REGION Network 38: ABFV 207 OPEN FB
   RUNG wire#powerrail
      { S7_Templates := "SrcType := Int" } EQ_Contact(in1 := "MODE SELECTION DB"."UF PLC_1 MODE BUFF", in2 := 1)
      { S7_Templates := "SrcType := Int" } EQ_Contact(in1 := "MODE SELECTION DB"."UF PLC_1 PROCESS BUFF", in2 := 870)
      Contact( "INPUT MAPPING DB"."ABFV-207 FEED BACK OPEN" )
      Move(in := 875, out1 => "MODE SELECTION DB"."UF PLC_1 PROCESS BUFF")
   END_RUNG
   // the same network as SCL:
   IF ("MODE SELECTION DB"."UF PLC_1 MODE BUFF" = 1) AND ("MODE SELECTION DB"."UF PLC_1 PROCESS BUFF" = 870) AND "INPUT MAPPING DB"."ABFV-207 FEED BACK OPEN" THEN
       "MODE SELECTION DB"."UF PLC_1 PROCESS BUFF" := 875;
   END_IF;
END_REGION

REGION Network 39: ABFV 208 OPEN FB
   RUNG wire#powerrail
      { S7_Templates := "SrcType := Int" } EQ_Contact(in1 := "MODE SELECTION DB"."UF PLC_1 MODE BUFF", in2 := 1)
      { S7_Templates := "SrcType := Int" } EQ_Contact(in1 := "MODE SELECTION DB"."UF PLC_1 PROCESS BUFF", in2 := 875)
      Contact( "INPUT MAPPING DB"."ABFV-208 FEED BACK OPEN" )
      { S7_Templates := "time_type := Time" } "IEC_Timer_0_DB_85".TON(pt := T#5s, et =>)
      Move(in := 880, out1 => "MODE SELECTION DB"."UF PLC_1 PROCESS BUFF")
   END_RUNG
   // the same network as SCL:
   "IEC_Timer_0_DB_85".TON(IN := ("MODE SELECTION DB"."UF PLC_1 MODE BUFF" = 1) AND ("MODE SELECTION DB"."UF PLC_1 PROCESS BUFF" = 875) AND "INPUT MAPPING DB"."ABFV-208 FEED BACK OPEN",
                           PT := T#5s);
   IF "IEC_Timer_0_DB_85".Q THEN "MODE SELECTION DB"."UF PLC_1 PROCESS BUFF" := 880; END_IF;
END_REGION

REGION Network 40: BACKWASH_1
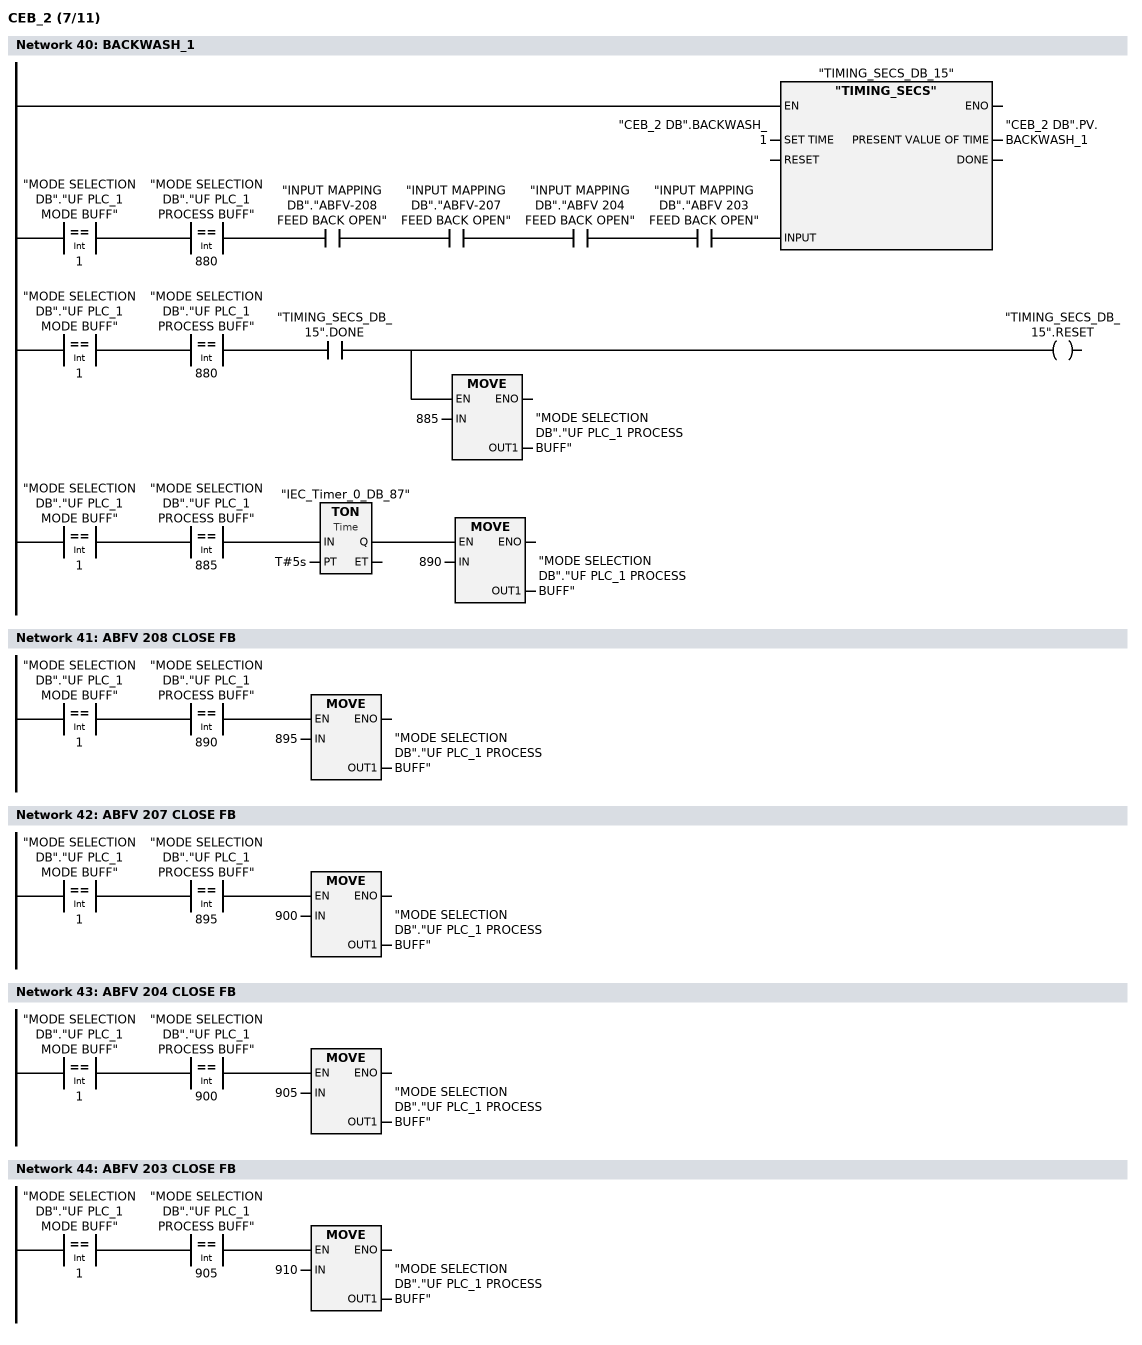
   RUNG wire#powerrail
      "TIMING_SECS_DB_15"(INPUT := wire#w1, "SET TIME" := "CEB_2 DB".BACKWASH_1, RESET :=, "PRESENT VALUE OF TIME" => "CEB_2 DB".PV.BACKWASH_1, DONE =>)
   END_RUNG
   RUNG wire#powerrail
      { S7_Templates := "SrcType := Int" } EQ_Contact(in1 := "MODE SELECTION DB"."UF PLC_1 MODE BUFF", in2 := 1)
      { S7_Templates := "SrcType := Int" } EQ_Contact(in1 := "MODE SELECTION DB"."UF PLC_1 PROCESS BUFF", in2 := 880)
      Contact( "INPUT MAPPING DB"."ABFV-208 FEED BACK OPEN" )
      Contact( "INPUT MAPPING DB"."ABFV-207 FEED BACK OPEN" )
      Contact( "INPUT MAPPING DB"."ABFV 204 FEED BACK OPEN" )
      Contact( "INPUT MAPPING DB"."ABFV 203 FEED BACK OPEN" )
   END_RUNG wire#w1
   RUNG wire#powerrail
      { S7_Templates := "SrcType := Int" } EQ_Contact(in1 := "MODE SELECTION DB"."UF PLC_1 MODE BUFF", in2 := 1)
      { S7_Templates := "SrcType := Int" } EQ_Contact(in1 := "MODE SELECTION DB"."UF PLC_1 PROCESS BUFF", in2 := 880)
      Contact( "TIMING_SECS_DB_15".DONE )
      wire#w2
      Coil( "TIMING_SECS_DB_15".RESET )
   END_RUNG
   RUNG wire#w2
      Move(in := 885, out1 => "MODE SELECTION DB"."UF PLC_1 PROCESS BUFF")
   END_RUNG
   RUNG wire#powerrail
      { S7_Templates := "SrcType := Int" } EQ_Contact(in1 := "MODE SELECTION DB"."UF PLC_1 MODE BUFF", in2 := 1)
      { S7_Templates := "SrcType := Int" } EQ_Contact(in1 := "MODE SELECTION DB"."UF PLC_1 PROCESS BUFF", in2 := 885)
      { S7_Templates := "time_type := Time" } "IEC_Timer_0_DB_87".TON(pt := T#5s, et =>)
      Move(in := 890, out1 => "MODE SELECTION DB"."UF PLC_1 PROCESS BUFF")
   END_RUNG
   // the same network as SCL:
   "TIMING_SECS_DB_15"("SET TIME" := "CEB_2 DB".BACKWASH_1,   // "TIMING_SECS"
                       INPUT := ("MODE SELECTION DB"."UF PLC_1 MODE BUFF" = 1) AND ("MODE SELECTION DB"."UF PLC_1 PROCESS BUFF" = 880) AND "INPUT MAPPING DB"."ABFV-208 FEED BACK OPEN" AND "INPUT MAPPING DB"."ABFV-207 FEED BACK OPEN" AND "INPUT MAPPING DB"."ABFV 204 FEED BACK OPEN" AND "INPUT MAPPING DB"."ABFV 203 FEED BACK OPEN",
                       "PRESENT VALUE OF TIME" => "CEB_2 DB".PV.BACKWASH_1);
   "TIMING_SECS_DB_15".RESET := ("MODE SELECTION DB"."UF PLC_1 MODE BUFF" = 1) AND ("MODE SELECTION DB"."UF PLC_1 PROCESS BUFF" = 880) AND "TIMING_SECS_DB_15".DONE;
   IF "TIMING_SECS_DB_15".RESET THEN "MODE SELECTION DB"."UF PLC_1 PROCESS BUFF" := 885; END_IF;
   "IEC_Timer_0_DB_87".TON(IN := ("MODE SELECTION DB"."UF PLC_1 MODE BUFF" = 1) AND ("MODE SELECTION DB"."UF PLC_1 PROCESS BUFF" = 885),
                           PT := T#5s);
   IF "IEC_Timer_0_DB_87".Q THEN "MODE SELECTION DB"."UF PLC_1 PROCESS BUFF" := 890; END_IF;
END_REGION

REGION Network 41: ABFV 208 CLOSE FB
   RUNG wire#powerrail
      { S7_Templates := "SrcType := Int" } EQ_Contact(in1 := "MODE SELECTION DB"."UF PLC_1 MODE BUFF", in2 := 1)
      { S7_Templates := "SrcType := Int" } EQ_Contact(in1 := "MODE SELECTION DB"."UF PLC_1 PROCESS BUFF", in2 := 890)
      Move(in := 895, out1 => "MODE SELECTION DB"."UF PLC_1 PROCESS BUFF")
   END_RUNG
   // the same network as SCL:
   IF ("MODE SELECTION DB"."UF PLC_1 MODE BUFF" = 1) AND ("MODE SELECTION DB"."UF PLC_1 PROCESS BUFF" = 890) THEN
       "MODE SELECTION DB"."UF PLC_1 PROCESS BUFF" := 895;
   END_IF;
END_REGION

REGION Network 42: ABFV 207 CLOSE FB
   RUNG wire#powerrail
      { S7_Templates := "SrcType := Int" } EQ_Contact(in1 := "MODE SELECTION DB"."UF PLC_1 MODE BUFF", in2 := 1)
      { S7_Templates := "SrcType := Int" } EQ_Contact(in1 := "MODE SELECTION DB"."UF PLC_1 PROCESS BUFF", in2 := 895)
      Move(in := 900, out1 => "MODE SELECTION DB"."UF PLC_1 PROCESS BUFF")
   END_RUNG
   // the same network as SCL:
   IF ("MODE SELECTION DB"."UF PLC_1 MODE BUFF" = 1) AND ("MODE SELECTION DB"."UF PLC_1 PROCESS BUFF" = 895) THEN
       "MODE SELECTION DB"."UF PLC_1 PROCESS BUFF" := 900;
   END_IF;
END_REGION

REGION Network 43: ABFV 204 CLOSE FB
   RUNG wire#powerrail
      { S7_Templates := "SrcType := Int" } EQ_Contact(in1 := "MODE SELECTION DB"."UF PLC_1 MODE BUFF", in2 := 1)
      { S7_Templates := "SrcType := Int" } EQ_Contact(in1 := "MODE SELECTION DB"."UF PLC_1 PROCESS BUFF", in2 := 900)
      Move(in := 905, out1 => "MODE SELECTION DB"."UF PLC_1 PROCESS BUFF")
   END_RUNG
   // the same network as SCL:
   IF ("MODE SELECTION DB"."UF PLC_1 MODE BUFF" = 1) AND ("MODE SELECTION DB"."UF PLC_1 PROCESS BUFF" = 900) THEN
       "MODE SELECTION DB"."UF PLC_1 PROCESS BUFF" := 905;
   END_IF;
END_REGION

REGION Network 44: ABFV 203 CLOSE FB
   RUNG wire#powerrail
      { S7_Templates := "SrcType := Int" } EQ_Contact(in1 := "MODE SELECTION DB"."UF PLC_1 MODE BUFF", in2 := 1)
      { S7_Templates := "SrcType := Int" } EQ_Contact(in1 := "MODE SELECTION DB"."UF PLC_1 PROCESS BUFF", in2 := 905)
      Move(in := 910, out1 => "MODE SELECTION DB"."UF PLC_1 PROCESS BUFF")
   END_RUNG
   // the same network as SCL:
   IF ("MODE SELECTION DB"."UF PLC_1 MODE BUFF" = 1) AND ("MODE SELECTION DB"."UF PLC_1 PROCESS BUFF" = 905) THEN
       "MODE SELECTION DB"."UF PLC_1 PROCESS BUFF" := 910;
   END_IF;
END_REGION

REGION Network 45: 915
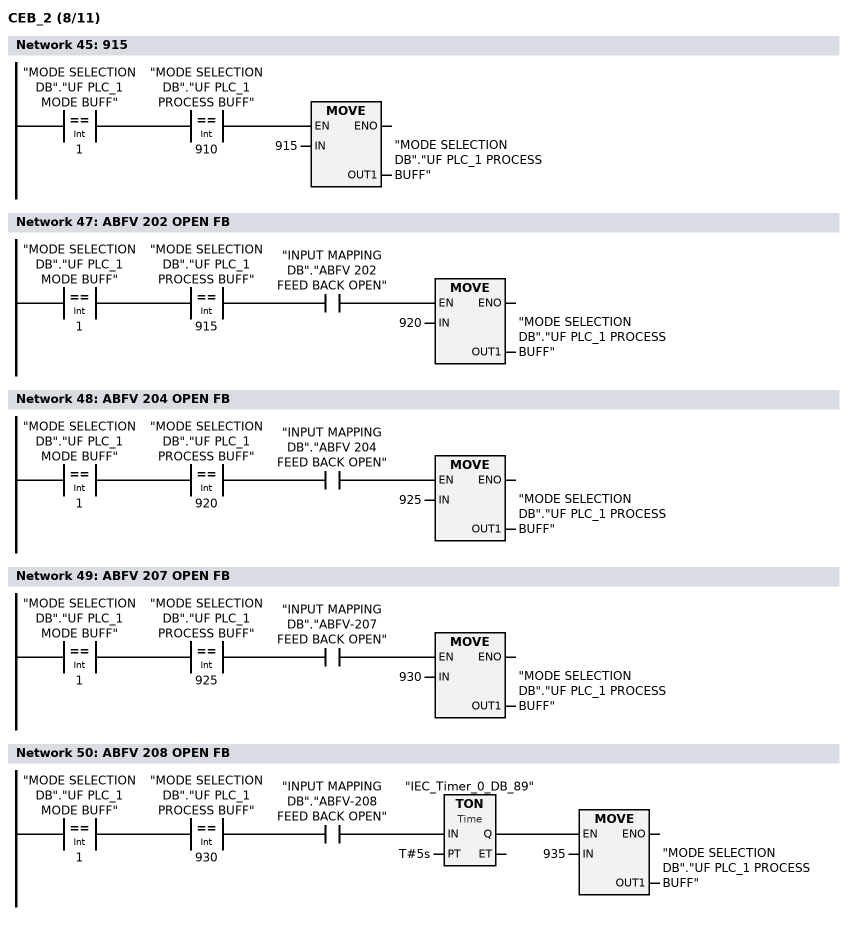
   RUNG wire#powerrail
      { S7_Templates := "SrcType := Int" } EQ_Contact(in1 := "MODE SELECTION DB"."UF PLC_1 MODE BUFF", in2 := 1)
      { S7_Templates := "SrcType := Int" } EQ_Contact(in1 := "MODE SELECTION DB"."UF PLC_1 PROCESS BUFF", in2 := 910)
      Move(in := 915, out1 => "MODE SELECTION DB"."UF PLC_1 PROCESS BUFF")
   END_RUNG
   // the same network as SCL:
   IF ("MODE SELECTION DB"."UF PLC_1 MODE BUFF" = 1) AND ("MODE SELECTION DB"."UF PLC_1 PROCESS BUFF" = 910) THEN
       "MODE SELECTION DB"."UF PLC_1 PROCESS BUFF" := 915;
   END_IF;
END_REGION

REGION Network 47: ABFV 202 OPEN FB
   RUNG wire#powerrail
      { S7_Templates := "SrcType := Int" } EQ_Contact(in1 := "MODE SELECTION DB"."UF PLC_1 MODE BUFF", in2 := 1)
      { S7_Templates := "SrcType := Int" } EQ_Contact(in1 := "MODE SELECTION DB"."UF PLC_1 PROCESS BUFF", in2 := 915)
      Contact( "INPUT MAPPING DB"."ABFV 202 FEED BACK OPEN" )
      Move(in := 920, out1 => "MODE SELECTION DB"."UF PLC_1 PROCESS BUFF")
   END_RUNG
   // the same network as SCL:
   IF ("MODE SELECTION DB"."UF PLC_1 MODE BUFF" = 1) AND ("MODE SELECTION DB"."UF PLC_1 PROCESS BUFF" = 915) AND "INPUT MAPPING DB"."ABFV 202 FEED BACK OPEN" THEN
       "MODE SELECTION DB"."UF PLC_1 PROCESS BUFF" := 920;
   END_IF;
END_REGION

REGION Network 48: ABFV 204 OPEN FB
   RUNG wire#powerrail
      { S7_Templates := "SrcType := Int" } EQ_Contact(in1 := "MODE SELECTION DB"."UF PLC_1 MODE BUFF", in2 := 1)
      { S7_Templates := "SrcType := Int" } EQ_Contact(in1 := "MODE SELECTION DB"."UF PLC_1 PROCESS BUFF", in2 := 920)
      Contact( "INPUT MAPPING DB"."ABFV 204 FEED BACK OPEN" )
      Move(in := 925, out1 => "MODE SELECTION DB"."UF PLC_1 PROCESS BUFF")
   END_RUNG
   // the same network as SCL:
   IF ("MODE SELECTION DB"."UF PLC_1 MODE BUFF" = 1) AND ("MODE SELECTION DB"."UF PLC_1 PROCESS BUFF" = 920) AND "INPUT MAPPING DB"."ABFV 204 FEED BACK OPEN" THEN
       "MODE SELECTION DB"."UF PLC_1 PROCESS BUFF" := 925;
   END_IF;
END_REGION

REGION Network 49: ABFV 207 OPEN FB
   RUNG wire#powerrail
      { S7_Templates := "SrcType := Int" } EQ_Contact(in1 := "MODE SELECTION DB"."UF PLC_1 MODE BUFF", in2 := 1)
      { S7_Templates := "SrcType := Int" } EQ_Contact(in1 := "MODE SELECTION DB"."UF PLC_1 PROCESS BUFF", in2 := 925)
      Contact( "INPUT MAPPING DB"."ABFV-207 FEED BACK OPEN" )
      Move(in := 930, out1 => "MODE SELECTION DB"."UF PLC_1 PROCESS BUFF")
   END_RUNG
   // the same network as SCL:
   IF ("MODE SELECTION DB"."UF PLC_1 MODE BUFF" = 1) AND ("MODE SELECTION DB"."UF PLC_1 PROCESS BUFF" = 925) AND "INPUT MAPPING DB"."ABFV-207 FEED BACK OPEN" THEN
       "MODE SELECTION DB"."UF PLC_1 PROCESS BUFF" := 930;
   END_IF;
END_REGION

REGION Network 50: ABFV 208 OPEN FB
   RUNG wire#powerrail
      { S7_Templates := "SrcType := Int" } EQ_Contact(in1 := "MODE SELECTION DB"."UF PLC_1 MODE BUFF", in2 := 1)
      { S7_Templates := "SrcType := Int" } EQ_Contact(in1 := "MODE SELECTION DB"."UF PLC_1 PROCESS BUFF", in2 := 930)
      Contact( "INPUT MAPPING DB"."ABFV-208 FEED BACK OPEN" )
      { S7_Templates := "time_type := Time" } "IEC_Timer_0_DB_89".TON(pt := T#5s, et =>)
      Move(in := 935, out1 => "MODE SELECTION DB"."UF PLC_1 PROCESS BUFF")
   END_RUNG
   // the same network as SCL:
   "IEC_Timer_0_DB_89".TON(IN := ("MODE SELECTION DB"."UF PLC_1 MODE BUFF" = 1) AND ("MODE SELECTION DB"."UF PLC_1 PROCESS BUFF" = 930) AND "INPUT MAPPING DB"."ABFV-208 FEED BACK OPEN",
                           PT := T#5s);
   IF "IEC_Timer_0_DB_89".Q THEN "MODE SELECTION DB"."UF PLC_1 PROCESS BUFF" := 935; END_IF;
END_REGION

REGION Network 51: BACKWASH_2
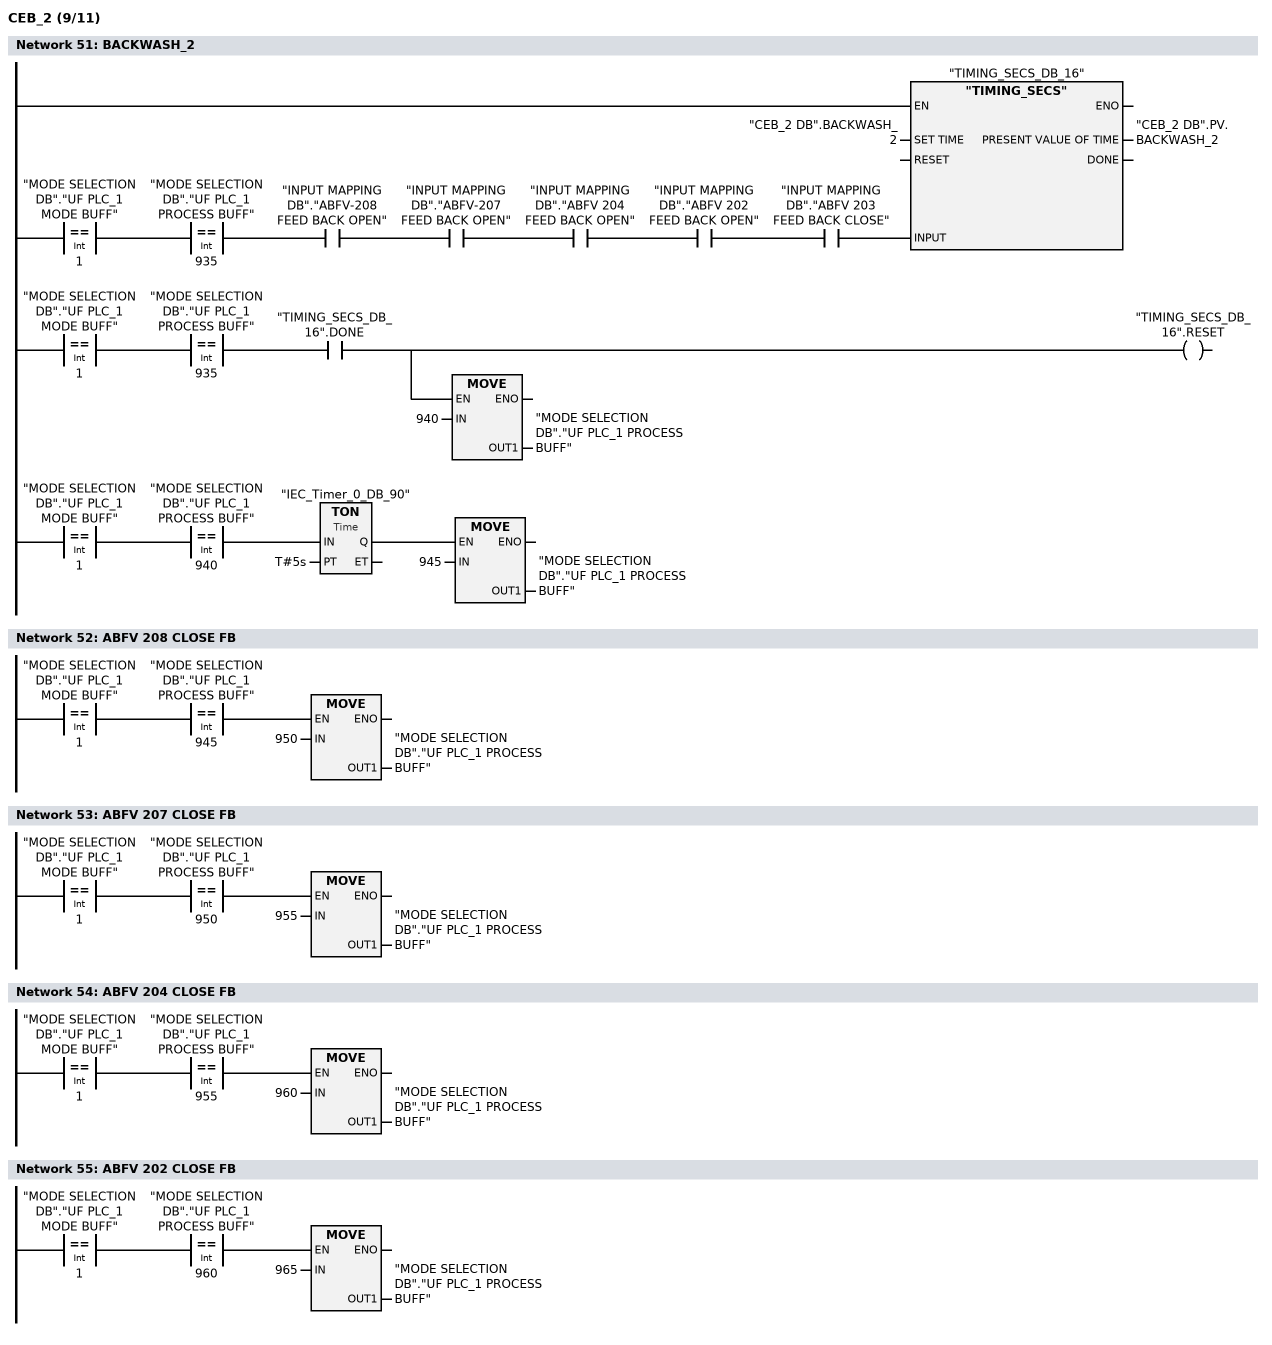
   RUNG wire#powerrail
      "TIMING_SECS_DB_16"(INPUT := wire#w1, "SET TIME" := "CEB_2 DB".BACKWASH_2, RESET :=, "PRESENT VALUE OF TIME" => "CEB_2 DB".PV.BACKWASH_2, DONE =>)
   END_RUNG
   RUNG wire#powerrail
      { S7_Templates := "SrcType := Int" } EQ_Contact(in1 := "MODE SELECTION DB"."UF PLC_1 MODE BUFF", in2 := 1)
      { S7_Templates := "SrcType := Int" } EQ_Contact(in1 := "MODE SELECTION DB"."UF PLC_1 PROCESS BUFF", in2 := 935)
      Contact( "INPUT MAPPING DB"."ABFV-208 FEED BACK OPEN" )
      Contact( "INPUT MAPPING DB"."ABFV-207 FEED BACK OPEN" )
      Contact( "INPUT MAPPING DB"."ABFV 204 FEED BACK OPEN" )
      Contact( "INPUT MAPPING DB"."ABFV 202 FEED BACK OPEN" )
      Contact( "INPUT MAPPING DB"."ABFV 203 FEED BACK CLOSE" )
   END_RUNG wire#w1
   RUNG wire#powerrail
      { S7_Templates := "SrcType := Int" } EQ_Contact(in1 := "MODE SELECTION DB"."UF PLC_1 MODE BUFF", in2 := 1)
      { S7_Templates := "SrcType := Int" } EQ_Contact(in1 := "MODE SELECTION DB"."UF PLC_1 PROCESS BUFF", in2 := 935)
      Contact( "TIMING_SECS_DB_16".DONE )
      wire#w2
      Coil( "TIMING_SECS_DB_16".RESET )
   END_RUNG
   RUNG wire#w2
      Move(in := 940, out1 => "MODE SELECTION DB"."UF PLC_1 PROCESS BUFF")
   END_RUNG
   RUNG wire#powerrail
      { S7_Templates := "SrcType := Int" } EQ_Contact(in1 := "MODE SELECTION DB"."UF PLC_1 MODE BUFF", in2 := 1)
      { S7_Templates := "SrcType := Int" } EQ_Contact(in1 := "MODE SELECTION DB"."UF PLC_1 PROCESS BUFF", in2 := 940)
      { S7_Templates := "time_type := Time" } "IEC_Timer_0_DB_90".TON(pt := T#5s, et =>)
      Move(in := 945, out1 => "MODE SELECTION DB"."UF PLC_1 PROCESS BUFF")
   END_RUNG
   // the same network as SCL:
   "TIMING_SECS_DB_16"("SET TIME" := "CEB_2 DB".BACKWASH_2,   // "TIMING_SECS"
                       INPUT := ("MODE SELECTION DB"."UF PLC_1 MODE BUFF" = 1) AND ("MODE SELECTION DB"."UF PLC_1 PROCESS BUFF" = 935) AND "INPUT MAPPING DB"."ABFV-208 FEED BACK OPEN" AND "INPUT MAPPING DB"."ABFV-207 FEED BACK OPEN" AND "INPUT MAPPING DB"."ABFV 204 FEED BACK OPEN" AND "INPUT MAPPING DB"."ABFV 202 FEED BACK OPEN" AND "INPUT MAPPING DB"."ABFV 203 FEED BACK CLOSE",
                       "PRESENT VALUE OF TIME" => "CEB_2 DB".PV.BACKWASH_2);
   "TIMING_SECS_DB_16".RESET := ("MODE SELECTION DB"."UF PLC_1 MODE BUFF" = 1) AND ("MODE SELECTION DB"."UF PLC_1 PROCESS BUFF" = 935) AND "TIMING_SECS_DB_16".DONE;
   IF "TIMING_SECS_DB_16".RESET THEN "MODE SELECTION DB"."UF PLC_1 PROCESS BUFF" := 940; END_IF;
   "IEC_Timer_0_DB_90".TON(IN := ("MODE SELECTION DB"."UF PLC_1 MODE BUFF" = 1) AND ("MODE SELECTION DB"."UF PLC_1 PROCESS BUFF" = 940),
                           PT := T#5s);
   IF "IEC_Timer_0_DB_90".Q THEN "MODE SELECTION DB"."UF PLC_1 PROCESS BUFF" := 945; END_IF;
END_REGION

REGION Network 52: ABFV 208 CLOSE FB
   RUNG wire#powerrail
      { S7_Templates := "SrcType := Int" } EQ_Contact(in1 := "MODE SELECTION DB"."UF PLC_1 MODE BUFF", in2 := 1)
      { S7_Templates := "SrcType := Int" } EQ_Contact(in1 := "MODE SELECTION DB"."UF PLC_1 PROCESS BUFF", in2 := 945)
      Move(in := 950, out1 => "MODE SELECTION DB"."UF PLC_1 PROCESS BUFF")
   END_RUNG
   // the same network as SCL:
   IF ("MODE SELECTION DB"."UF PLC_1 MODE BUFF" = 1) AND ("MODE SELECTION DB"."UF PLC_1 PROCESS BUFF" = 945) THEN
       "MODE SELECTION DB"."UF PLC_1 PROCESS BUFF" := 950;
   END_IF;
END_REGION

REGION Network 53: ABFV 207 CLOSE FB
   RUNG wire#powerrail
      { S7_Templates := "SrcType := Int" } EQ_Contact(in1 := "MODE SELECTION DB"."UF PLC_1 MODE BUFF", in2 := 1)
      { S7_Templates := "SrcType := Int" } EQ_Contact(in1 := "MODE SELECTION DB"."UF PLC_1 PROCESS BUFF", in2 := 950)
      Move(in := 955, out1 => "MODE SELECTION DB"."UF PLC_1 PROCESS BUFF")
   END_RUNG
   // the same network as SCL:
   IF ("MODE SELECTION DB"."UF PLC_1 MODE BUFF" = 1) AND ("MODE SELECTION DB"."UF PLC_1 PROCESS BUFF" = 950) THEN
       "MODE SELECTION DB"."UF PLC_1 PROCESS BUFF" := 955;
   END_IF;
END_REGION

REGION Network 54: ABFV 204 CLOSE FB
   RUNG wire#powerrail
      { S7_Templates := "SrcType := Int" } EQ_Contact(in1 := "MODE SELECTION DB"."UF PLC_1 MODE BUFF", in2 := 1)
      { S7_Templates := "SrcType := Int" } EQ_Contact(in1 := "MODE SELECTION DB"."UF PLC_1 PROCESS BUFF", in2 := 955)
      Move(in := 960, out1 => "MODE SELECTION DB"."UF PLC_1 PROCESS BUFF")
   END_RUNG
   // the same network as SCL:
   IF ("MODE SELECTION DB"."UF PLC_1 MODE BUFF" = 1) AND ("MODE SELECTION DB"."UF PLC_1 PROCESS BUFF" = 955) THEN
       "MODE SELECTION DB"."UF PLC_1 PROCESS BUFF" := 960;
   END_IF;
END_REGION

REGION Network 55: ABFV 202 CLOSE FB
   RUNG wire#powerrail
      { S7_Templates := "SrcType := Int" } EQ_Contact(in1 := "MODE SELECTION DB"."UF PLC_1 MODE BUFF", in2 := 1)
      { S7_Templates := "SrcType := Int" } EQ_Contact(in1 := "MODE SELECTION DB"."UF PLC_1 PROCESS BUFF", in2 := 960)
      Move(in := 965, out1 => "MODE SELECTION DB"."UF PLC_1 PROCESS BUFF")
   END_RUNG
   // the same network as SCL:
   IF ("MODE SELECTION DB"."UF PLC_1 MODE BUFF" = 1) AND ("MODE SELECTION DB"."UF PLC_1 PROCESS BUFF" = 960) THEN
       "MODE SELECTION DB"."UF PLC_1 PROCESS BUFF" := 965;
   END_IF;
END_REGION

REGION Network 56: 970
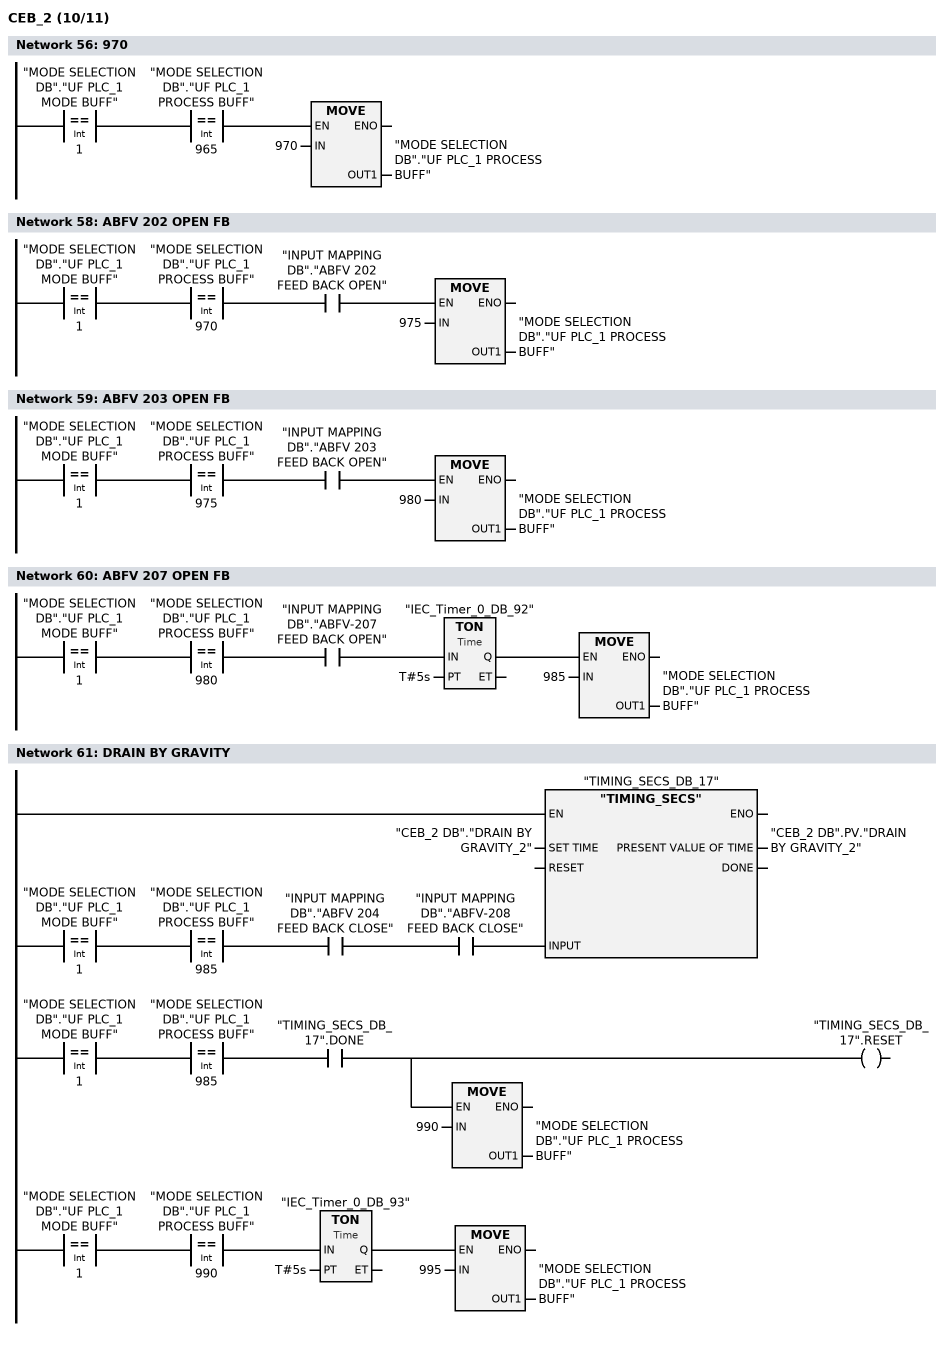
   RUNG wire#powerrail
      { S7_Templates := "SrcType := Int" } EQ_Contact(in1 := "MODE SELECTION DB"."UF PLC_1 MODE BUFF", in2 := 1)
      { S7_Templates := "SrcType := Int" } EQ_Contact(in1 := "MODE SELECTION DB"."UF PLC_1 PROCESS BUFF", in2 := 965)
      Move(in := 970, out1 => "MODE SELECTION DB"."UF PLC_1 PROCESS BUFF")
   END_RUNG
   // the same network as SCL:
   IF ("MODE SELECTION DB"."UF PLC_1 MODE BUFF" = 1) AND ("MODE SELECTION DB"."UF PLC_1 PROCESS BUFF" = 965) THEN
       "MODE SELECTION DB"."UF PLC_1 PROCESS BUFF" := 970;
   END_IF;
END_REGION

REGION Network 58: ABFV 202 OPEN FB
   RUNG wire#powerrail
      { S7_Templates := "SrcType := Int" } EQ_Contact(in1 := "MODE SELECTION DB"."UF PLC_1 MODE BUFF", in2 := 1)
      { S7_Templates := "SrcType := Int" } EQ_Contact(in1 := "MODE SELECTION DB"."UF PLC_1 PROCESS BUFF", in2 := 970)
      Contact( "INPUT MAPPING DB"."ABFV 202 FEED BACK OPEN" )
      Move(in := 975, out1 => "MODE SELECTION DB"."UF PLC_1 PROCESS BUFF")
   END_RUNG
   // the same network as SCL:
   IF ("MODE SELECTION DB"."UF PLC_1 MODE BUFF" = 1) AND ("MODE SELECTION DB"."UF PLC_1 PROCESS BUFF" = 970) AND "INPUT MAPPING DB"."ABFV 202 FEED BACK OPEN" THEN
       "MODE SELECTION DB"."UF PLC_1 PROCESS BUFF" := 975;
   END_IF;
END_REGION

REGION Network 59: ABFV 203 OPEN FB
   RUNG wire#powerrail
      { S7_Templates := "SrcType := Int" } EQ_Contact(in1 := "MODE SELECTION DB"."UF PLC_1 MODE BUFF", in2 := 1)
      { S7_Templates := "SrcType := Int" } EQ_Contact(in1 := "MODE SELECTION DB"."UF PLC_1 PROCESS BUFF", in2 := 975)
      Contact( "INPUT MAPPING DB"."ABFV 203 FEED BACK OPEN" )
      Move(in := 980, out1 => "MODE SELECTION DB"."UF PLC_1 PROCESS BUFF")
   END_RUNG
   // the same network as SCL:
   IF ("MODE SELECTION DB"."UF PLC_1 MODE BUFF" = 1) AND ("MODE SELECTION DB"."UF PLC_1 PROCESS BUFF" = 975) AND "INPUT MAPPING DB"."ABFV 203 FEED BACK OPEN" THEN
       "MODE SELECTION DB"."UF PLC_1 PROCESS BUFF" := 980;
   END_IF;
END_REGION

REGION Network 60: ABFV 207 OPEN FB
   RUNG wire#powerrail
      { S7_Templates := "SrcType := Int" } EQ_Contact(in1 := "MODE SELECTION DB"."UF PLC_1 MODE BUFF", in2 := 1)
      { S7_Templates := "SrcType := Int" } EQ_Contact(in1 := "MODE SELECTION DB"."UF PLC_1 PROCESS BUFF", in2 := 980)
      Contact( "INPUT MAPPING DB"."ABFV-207 FEED BACK OPEN" )
      { S7_Templates := "time_type := Time" } "IEC_Timer_0_DB_92".TON(pt := T#5s, et =>)
      Move(in := 985, out1 => "MODE SELECTION DB"."UF PLC_1 PROCESS BUFF")
   END_RUNG
   // the same network as SCL:
   "IEC_Timer_0_DB_92".TON(IN := ("MODE SELECTION DB"."UF PLC_1 MODE BUFF" = 1) AND ("MODE SELECTION DB"."UF PLC_1 PROCESS BUFF" = 980) AND "INPUT MAPPING DB"."ABFV-207 FEED BACK OPEN",
                           PT := T#5s);
   IF "IEC_Timer_0_DB_92".Q THEN "MODE SELECTION DB"."UF PLC_1 PROCESS BUFF" := 985; END_IF;
END_REGION

REGION Network 61: DRAIN BY GRAVITY
   RUNG wire#powerrail
      "TIMING_SECS_DB_17"(INPUT := wire#w1, "SET TIME" := "CEB_2 DB"."DRAIN BY GRAVITY_2", RESET :=, "PRESENT VALUE OF TIME" => "CEB_2 DB".PV."DRAIN BY GRAVITY_2", DONE =>)
   END_RUNG
   RUNG wire#powerrail
      { S7_Templates := "SrcType := Int" } EQ_Contact(in1 := "MODE SELECTION DB"."UF PLC_1 MODE BUFF", in2 := 1)
      { S7_Templates := "SrcType := Int" } EQ_Contact(in1 := "MODE SELECTION DB"."UF PLC_1 PROCESS BUFF", in2 := 985)
      Contact( "INPUT MAPPING DB"."ABFV 204 FEED BACK CLOSE" )
      Contact( "INPUT MAPPING DB"."ABFV-208 FEED BACK CLOSE" )
   END_RUNG wire#w1
   RUNG wire#powerrail
      { S7_Templates := "SrcType := Int" } EQ_Contact(in1 := "MODE SELECTION DB"."UF PLC_1 MODE BUFF", in2 := 1)
      { S7_Templates := "SrcType := Int" } EQ_Contact(in1 := "MODE SELECTION DB"."UF PLC_1 PROCESS BUFF", in2 := 985)
      Contact( "TIMING_SECS_DB_17".DONE )
      wire#w2
      Coil( "TIMING_SECS_DB_17".RESET )
   END_RUNG
   RUNG wire#w2
      Move(in := 990, out1 => "MODE SELECTION DB"."UF PLC_1 PROCESS BUFF")
   END_RUNG
   RUNG wire#powerrail
      { S7_Templates := "SrcType := Int" } EQ_Contact(in1 := "MODE SELECTION DB"."UF PLC_1 MODE BUFF", in2 := 1)
      { S7_Templates := "SrcType := Int" } EQ_Contact(in1 := "MODE SELECTION DB"."UF PLC_1 PROCESS BUFF", in2 := 990)
      { S7_Templates := "time_type := Time" } "IEC_Timer_0_DB_93".TON(pt := T#5s, et =>)
      Move(in := 995, out1 => "MODE SELECTION DB"."UF PLC_1 PROCESS BUFF")
   END_RUNG
   // the same network as SCL:
   "TIMING_SECS_DB_17"("SET TIME" := "CEB_2 DB"."DRAIN BY GRAVITY_2",   // "TIMING_SECS"
                       INPUT := ("MODE SELECTION DB"."UF PLC_1 MODE BUFF" = 1) AND ("MODE SELECTION DB"."UF PLC_1 PROCESS BUFF" = 985) AND "INPUT MAPPING DB"."ABFV 204 FEED BACK CLOSE" AND "INPUT MAPPING DB"."ABFV-208 FEED BACK CLOSE",
                       "PRESENT VALUE OF TIME" => "CEB_2 DB".PV."DRAIN BY GRAVITY_2");
   "TIMING_SECS_DB_17".RESET := ("MODE SELECTION DB"."UF PLC_1 MODE BUFF" = 1) AND ("MODE SELECTION DB"."UF PLC_1 PROCESS BUFF" = 985) AND "TIMING_SECS_DB_17".DONE;
   IF "TIMING_SECS_DB_17".RESET THEN "MODE SELECTION DB"."UF PLC_1 PROCESS BUFF" := 990; END_IF;
   "IEC_Timer_0_DB_93".TON(IN := ("MODE SELECTION DB"."UF PLC_1 MODE BUFF" = 1) AND ("MODE SELECTION DB"."UF PLC_1 PROCESS BUFF" = 990),
                           PT := T#5s);
   IF "IEC_Timer_0_DB_93".Q THEN "MODE SELECTION DB"."UF PLC_1 PROCESS BUFF" := 995; END_IF;
END_REGION

REGION Network 62: ABFV 207 CLOSE FB
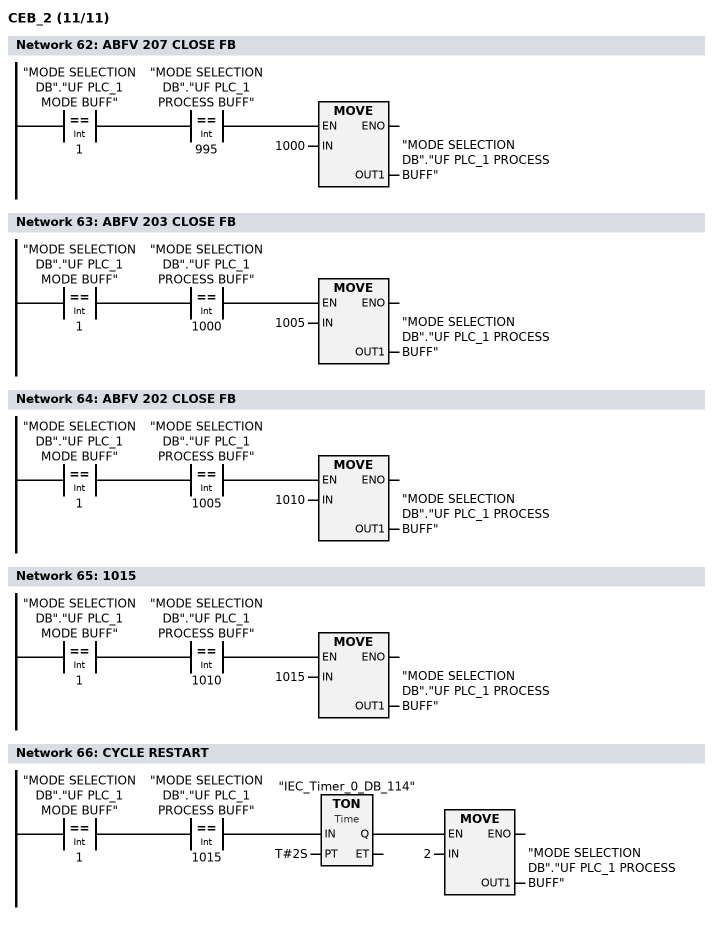
   RUNG wire#powerrail
      { S7_Templates := "SrcType := Int" } EQ_Contact(in1 := "MODE SELECTION DB"."UF PLC_1 MODE BUFF", in2 := 1)
      { S7_Templates := "SrcType := Int" } EQ_Contact(in1 := "MODE SELECTION DB"."UF PLC_1 PROCESS BUFF", in2 := 995)
      Move(in := 1000, out1 => "MODE SELECTION DB"."UF PLC_1 PROCESS BUFF")
   END_RUNG
   // the same network as SCL:
   IF ("MODE SELECTION DB"."UF PLC_1 MODE BUFF" = 1) AND ("MODE SELECTION DB"."UF PLC_1 PROCESS BUFF" = 995) THEN
       "MODE SELECTION DB"."UF PLC_1 PROCESS BUFF" := 1000;
   END_IF;
END_REGION

REGION Network 63: ABFV 203 CLOSE FB
   RUNG wire#powerrail
      { S7_Templates := "SrcType := Int" } EQ_Contact(in1 := "MODE SELECTION DB"."UF PLC_1 MODE BUFF", in2 := 1)
      { S7_Templates := "SrcType := Int" } EQ_Contact(in1 := "MODE SELECTION DB"."UF PLC_1 PROCESS BUFF", in2 := 1000)
      Move(in := 1005, out1 => "MODE SELECTION DB"."UF PLC_1 PROCESS BUFF")
   END_RUNG
   // the same network as SCL:
   IF ("MODE SELECTION DB"."UF PLC_1 MODE BUFF" = 1) AND ("MODE SELECTION DB"."UF PLC_1 PROCESS BUFF" = 1000) THEN
       "MODE SELECTION DB"."UF PLC_1 PROCESS BUFF" := 1005;
   END_IF;
END_REGION

REGION Network 64: ABFV 202 CLOSE FB
   RUNG wire#powerrail
      { S7_Templates := "SrcType := Int" } EQ_Contact(in1 := "MODE SELECTION DB"."UF PLC_1 MODE BUFF", in2 := 1)
      { S7_Templates := "SrcType := Int" } EQ_Contact(in1 := "MODE SELECTION DB"."UF PLC_1 PROCESS BUFF", in2 := 1005)
      Move(in := 1010, out1 => "MODE SELECTION DB"."UF PLC_1 PROCESS BUFF")
   END_RUNG
   // the same network as SCL:
   IF ("MODE SELECTION DB"."UF PLC_1 MODE BUFF" = 1) AND ("MODE SELECTION DB"."UF PLC_1 PROCESS BUFF" = 1005) THEN
       "MODE SELECTION DB"."UF PLC_1 PROCESS BUFF" := 1010;
   END_IF;
END_REGION

REGION Network 65: 1015
   RUNG wire#powerrail
      { S7_Templates := "SrcType := Int" } EQ_Contact(in1 := "MODE SELECTION DB"."UF PLC_1 MODE BUFF", in2 := 1)
      { S7_Templates := "SrcType := Int" } EQ_Contact(in1 := "MODE SELECTION DB"."UF PLC_1 PROCESS BUFF", in2 := 1010)
      Move(in := 1015, out1 => "MODE SELECTION DB"."UF PLC_1 PROCESS BUFF")
   END_RUNG
   // the same network as SCL:
   IF ("MODE SELECTION DB"."UF PLC_1 MODE BUFF" = 1) AND ("MODE SELECTION DB"."UF PLC_1 PROCESS BUFF" = 1010) THEN
       "MODE SELECTION DB"."UF PLC_1 PROCESS BUFF" := 1015;
   END_IF;
END_REGION

REGION Network 66: CYCLE RESTART
   RUNG wire#powerrail
      { S7_Templates := "SrcType := Int" } EQ_Contact(in1 := "MODE SELECTION DB"."UF PLC_1 MODE BUFF", in2 := 1)
      { S7_Templates := "SrcType := Int" } EQ_Contact(in1 := "MODE SELECTION DB"."UF PLC_1 PROCESS BUFF", in2 := 1015)
      { S7_Templates := "time_type := Time" } "IEC_Timer_0_DB_114".TON(pt := T#2S, et =>)
      Move(in := 2, out1 => "MODE SELECTION DB"."UF PLC_1 PROCESS BUFF")
   END_RUNG
   // the same network as SCL:
   "IEC_Timer_0_DB_114".TON(IN := ("MODE SELECTION DB"."UF PLC_1 MODE BUFF" = 1) AND ("MODE SELECTION DB"."UF PLC_1 PROCESS BUFF" = 1015),
                           PT := T#2S);
   IF "IEC_Timer_0_DB_114".Q THEN "MODE SELECTION DB"."UF PLC_1 PROCESS BUFF" := 2; END_IF;
END_REGION
END_FUNCTION

FUNCTION "AO SCALING" : Void   // FC17, LAD
{ S7_Optimized_Access := 'TRUE' }
// stored: SetENOAutomatically false
   VAR_TEMP   // added for the SCL form of the ladder/FBD networks
      _w1 : Bool;
   END_VAR
BEGIN

REGION Network 1: VFD P-502A
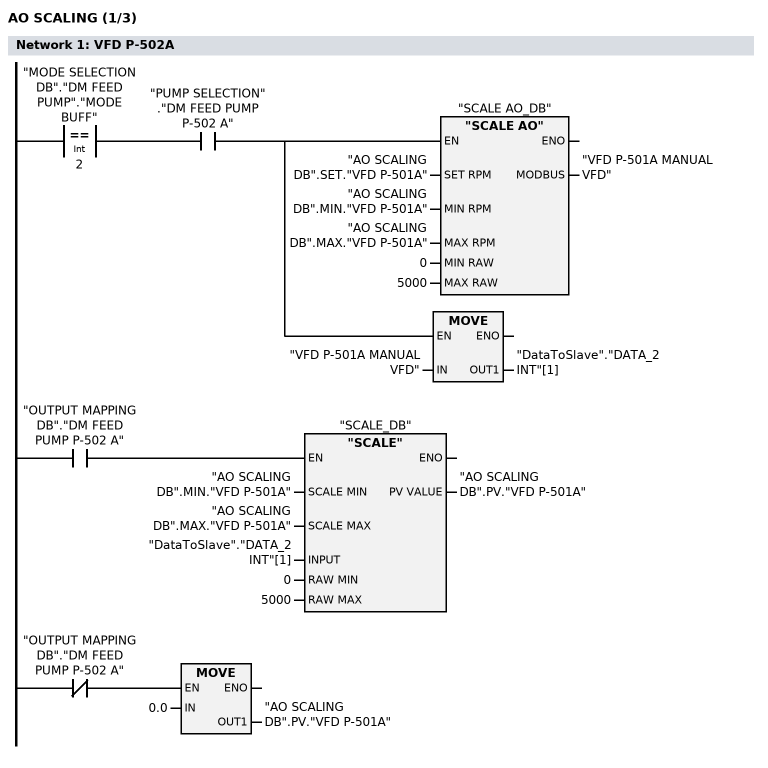
   RUNG wire#powerrail
      { S7_Templates := "SrcType := Int" } EQ_Contact(in1 := "MODE SELECTION DB"."DM FEED PUMP"."MODE BUFF", in2 := 2)
      Contact( "PUMP SELECTION"."DM FEED PUMP P-502 A" )
      wire#w1
      "SCALE AO_DB"("SET RPM" := "AO SCALING DB".SET."VFD P-501A", "MIN RPM" := "AO SCALING DB".MIN."VFD P-501A", "MAX RPM" := "AO SCALING DB".MAX."VFD P-501A", "MIN RAW" := 0, "MAX RAW" := 5000, MODBUS => "VFD P-501A MANUAL VFD")
   END_RUNG
   RUNG wire#w1
      Move(in := "VFD P-501A MANUAL VFD", out1 => "DataToSlave"."DATA_2 INT"[1])
   END_RUNG
   RUNG wire#powerrail
      Contact( "OUTPUT MAPPING DB"."DM FEED PUMP P-502 A" )
      "SCALE_DB"("SCALE MIN" := "AO SCALING DB".MIN."VFD P-501A", "SCALE MAX" := "AO SCALING DB".MAX."VFD P-501A", INPUT := "DataToSlave"."DATA_2 INT"[1], "RAW MIN" := 0, "RAW MAX" := 5000, "PV VALUE" => "AO SCALING DB".PV."VFD P-501A")
   END_RUNG
   RUNG wire#powerrail
      I_Contact( "OUTPUT MAPPING DB"."DM FEED PUMP P-502 A" )
      Move(in := 0.0, out1 => "AO SCALING DB".PV."VFD P-501A")
   END_RUNG
   // the same network as SCL:
   #_w1 := ("MODE SELECTION DB"."DM FEED PUMP"."MODE BUFF" = 2) AND "PUMP SELECTION"."DM FEED PUMP P-502 A";
   IF #_w1 THEN
       "SCALE AO_DB"("SET RPM" := "AO SCALING DB".SET."VFD P-501A",   // "SCALE AO"
                     "MIN RPM" := "AO SCALING DB".MIN."VFD P-501A",
                     "MAX RPM" := "AO SCALING DB".MAX."VFD P-501A",
                     "MIN RAW" := 0,
                     "MAX RAW" := 5000,
                     MODBUS => "VFD P-501A MANUAL VFD");
       "DataToSlave"."DATA_2 INT"[1] := "VFD P-501A MANUAL VFD";
   END_IF;
   IF "OUTPUT MAPPING DB"."DM FEED PUMP P-502 A" THEN
       "SCALE_DB"("SCALE MIN" := "AO SCALING DB".MIN."VFD P-501A",   // "SCALE"
                  "SCALE MAX" := "AO SCALING DB".MAX."VFD P-501A",
                  INPUT := "DataToSlave"."DATA_2 INT"[1],
                  "RAW MIN" := 0,
                  "RAW MAX" := 5000,
                  "PV VALUE" => "AO SCALING DB".PV."VFD P-501A");
   END_IF;
   IF NOT "OUTPUT MAPPING DB"."DM FEED PUMP P-502 A" THEN "AO SCALING DB".PV."VFD P-501A" := 0.0; END_IF;
END_REGION

REGION Network 2: VFD P-502B
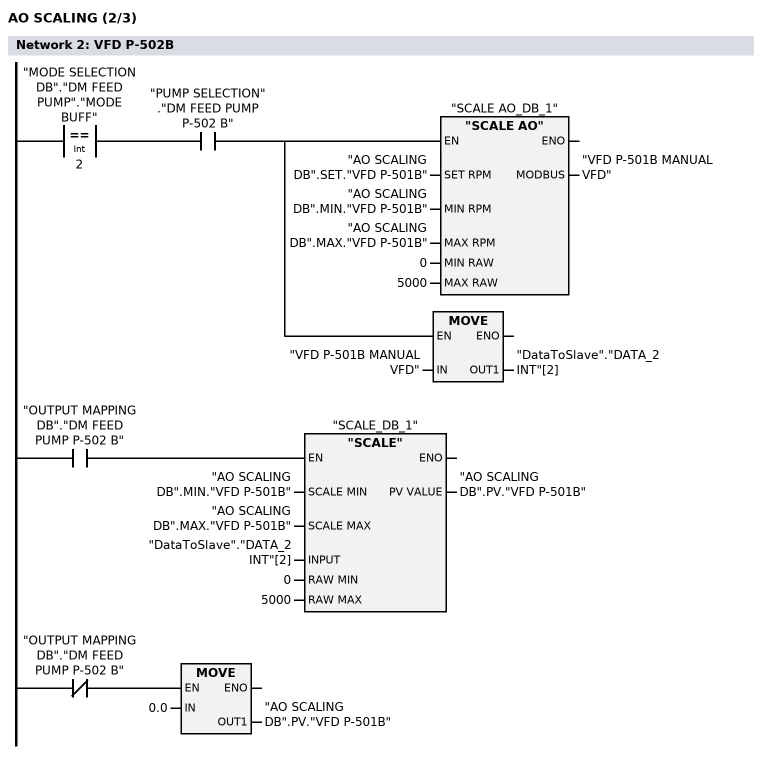
   RUNG wire#powerrail
      { S7_Templates := "SrcType := Int" } EQ_Contact(in1 := "MODE SELECTION DB"."DM FEED PUMP"."MODE BUFF", in2 := 2)
      Contact( "PUMP SELECTION"."DM FEED PUMP P-502 B" )
      wire#w1
      "SCALE AO_DB_1"("SET RPM" := "AO SCALING DB".SET."VFD P-501B", "MIN RPM" := "AO SCALING DB".MIN."VFD P-501B", "MAX RPM" := "AO SCALING DB".MAX."VFD P-501B", "MIN RAW" := 0, "MAX RAW" := 5000, MODBUS => "VFD P-501B MANUAL VFD")
   END_RUNG
   RUNG wire#w1
      Move(in := "VFD P-501B MANUAL VFD", out1 => "DataToSlave"."DATA_2 INT"[2])
   END_RUNG
   RUNG wire#powerrail
      Contact( "OUTPUT MAPPING DB"."DM FEED PUMP P-502 B" )
      "SCALE_DB_1"("SCALE MIN" := "AO SCALING DB".MIN."VFD P-501B", "SCALE MAX" := "AO SCALING DB".MAX."VFD P-501B", INPUT := "DataToSlave"."DATA_2 INT"[2], "RAW MIN" := 0, "RAW MAX" := 5000, "PV VALUE" => "AO SCALING DB".PV."VFD P-501B")
   END_RUNG
   RUNG wire#powerrail
      I_Contact( "OUTPUT MAPPING DB"."DM FEED PUMP P-502 B" )
      Move(in := 0.0, out1 => "AO SCALING DB".PV."VFD P-501B")
   END_RUNG
   // the same network as SCL:
   #_w1 := ("MODE SELECTION DB"."DM FEED PUMP"."MODE BUFF" = 2) AND "PUMP SELECTION"."DM FEED PUMP P-502 B";
   IF #_w1 THEN
       "SCALE AO_DB_1"("SET RPM" := "AO SCALING DB".SET."VFD P-501B",   // "SCALE AO"
                       "MIN RPM" := "AO SCALING DB".MIN."VFD P-501B",
                       "MAX RPM" := "AO SCALING DB".MAX."VFD P-501B",
                       "MIN RAW" := 0,
                       "MAX RAW" := 5000,
                       MODBUS => "VFD P-501B MANUAL VFD");
       "DataToSlave"."DATA_2 INT"[2] := "VFD P-501B MANUAL VFD";
   END_IF;
   IF "OUTPUT MAPPING DB"."DM FEED PUMP P-502 B" THEN
       "SCALE_DB_1"("SCALE MIN" := "AO SCALING DB".MIN."VFD P-501B",   // "SCALE"
                    "SCALE MAX" := "AO SCALING DB".MAX."VFD P-501B",
                    INPUT := "DataToSlave"."DATA_2 INT"[2],
                    "RAW MIN" := 0,
                    "RAW MAX" := 5000,
                    "PV VALUE" => "AO SCALING DB".PV."VFD P-501B");
   END_IF;
   IF NOT "OUTPUT MAPPING DB"."DM FEED PUMP P-502 B" THEN "AO SCALING DB".PV."VFD P-501B" := 0.0; END_IF;
END_REGION

REGION Network 3: VFD P-502C
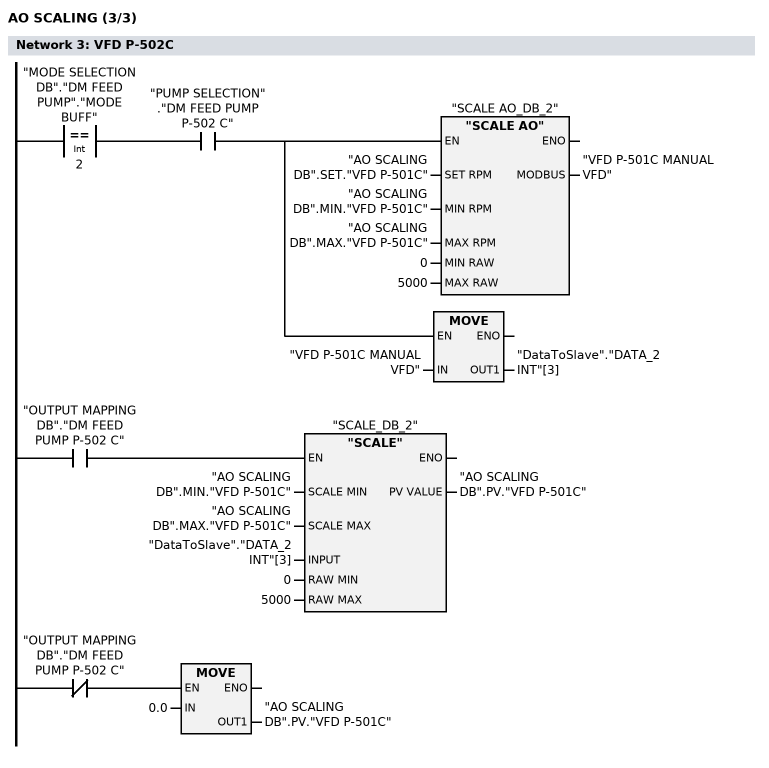
   RUNG wire#powerrail
      { S7_Templates := "SrcType := Int" } EQ_Contact(in1 := "MODE SELECTION DB"."DM FEED PUMP"."MODE BUFF", in2 := 2)
      Contact( "PUMP SELECTION"."DM FEED PUMP P-502 C" )
      wire#w1
      "SCALE AO_DB_2"("SET RPM" := "AO SCALING DB".SET."VFD P-501C", "MIN RPM" := "AO SCALING DB".MIN."VFD P-501C", "MAX RPM" := "AO SCALING DB".MAX."VFD P-501C", "MIN RAW" := 0, "MAX RAW" := 5000, MODBUS => "VFD P-501C MANUAL VFD")
   END_RUNG
   RUNG wire#w1
      Move(in := "VFD P-501C MANUAL VFD", out1 => "DataToSlave"."DATA_2 INT"[3])
   END_RUNG
   RUNG wire#powerrail
      Contact( "OUTPUT MAPPING DB"."DM FEED PUMP P-502 C" )
      "SCALE_DB_2"("SCALE MIN" := "AO SCALING DB".MIN."VFD P-501C", "SCALE MAX" := "AO SCALING DB".MAX."VFD P-501C", INPUT := "DataToSlave"."DATA_2 INT"[3], "RAW MIN" := 0, "RAW MAX" := 5000, "PV VALUE" => "AO SCALING DB".PV."VFD P-501C")
   END_RUNG
   RUNG wire#powerrail
      I_Contact( "OUTPUT MAPPING DB"."DM FEED PUMP P-502 C" )
      Move(in := 0.0, out1 => "AO SCALING DB".PV."VFD P-501C")
   END_RUNG
   // the same network as SCL:
   #_w1 := ("MODE SELECTION DB"."DM FEED PUMP"."MODE BUFF" = 2) AND "PUMP SELECTION"."DM FEED PUMP P-502 C";
   IF #_w1 THEN
       "SCALE AO_DB_2"("SET RPM" := "AO SCALING DB".SET."VFD P-501C",   // "SCALE AO"
                       "MIN RPM" := "AO SCALING DB".MIN."VFD P-501C",
                       "MAX RPM" := "AO SCALING DB".MAX."VFD P-501C",
                       "MIN RAW" := 0,
                       "MAX RAW" := 5000,
                       MODBUS => "VFD P-501C MANUAL VFD");
       "DataToSlave"."DATA_2 INT"[3] := "VFD P-501C MANUAL VFD";
   END_IF;
   IF "OUTPUT MAPPING DB"."DM FEED PUMP P-502 C" THEN
       "SCALE_DB_2"("SCALE MIN" := "AO SCALING DB".MIN."VFD P-501C",   // "SCALE"
                    "SCALE MAX" := "AO SCALING DB".MAX."VFD P-501C",
                    INPUT := "DataToSlave"."DATA_2 INT"[3],
                    "RAW MIN" := 0,
                    "RAW MAX" := 5000,
                    "PV VALUE" => "AO SCALING DB".PV."VFD P-501C");
   END_IF;
   IF NOT "OUTPUT MAPPING DB"."DM FEED PUMP P-502 C" THEN "AO SCALING DB".PV."VFD P-501C" := 0.0; END_IF;
END_REGION
END_FUNCTION

ORGANIZATION_BLOCK "PID P-502"   // OB30, LAD, CyclicInterrupt
{ S7_Optimized_Access := 'TRUE' }
// stored: SetENOAutomatically false
   VAR_INPUT
      Initial_Call : Bool;   // Initial call of this OB
      Event_Count : Int;   // Events discarded
   END_VAR
BEGIN

REGION Network 1: enable mode
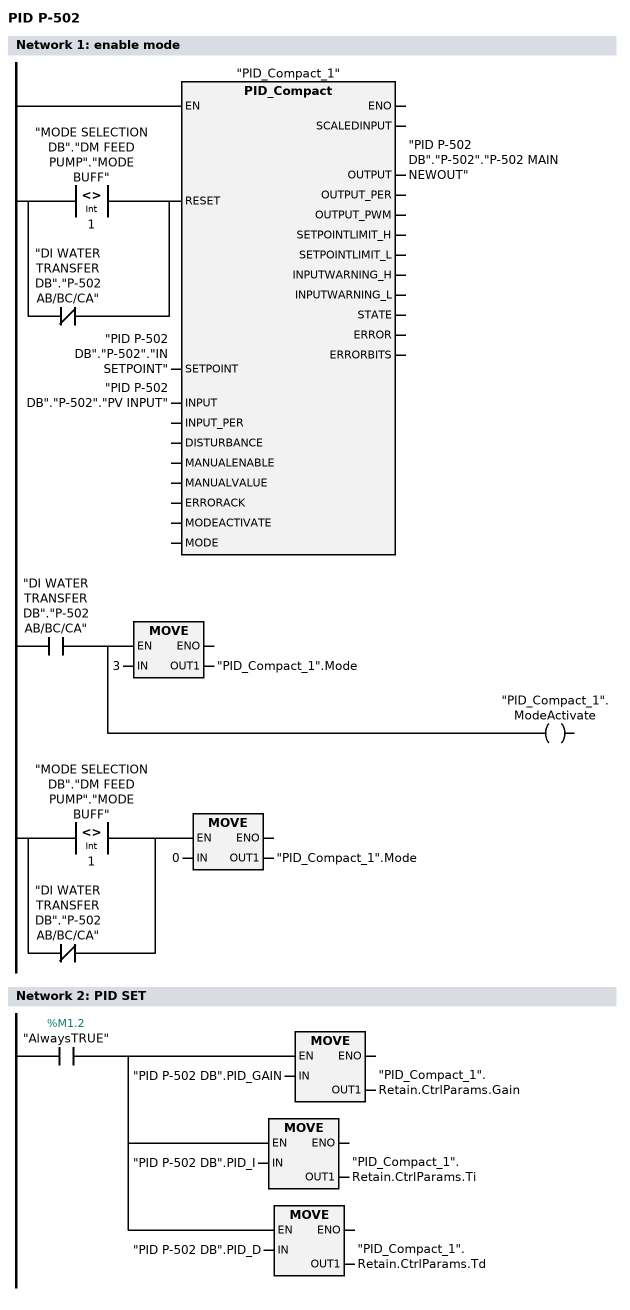
   RUNG wire#powerrail
      "PID_Compact_1".PID_Compact(Reset := wire#w1, Setpoint := "PID P-502 DB"."P-502"."IN SETPOINT", Input := "PID P-502 DB"."P-502"."PV INPUT", Input_PER :=, Disturbance :=, ManualEnable :=, ManualValue :=, ErrorAck :=, ModeActivate :=, Mode :=, ScaledInput =>, Output => "PID P-502 DB"."P-502"."P-502 MAIN NEWOUT", Output_PER =>, Output_PWM =>, SetpointLimit_H =>, SetpointLimit_L =>, InputWarning_H =>, InputWarning_L =>, State =>, Error =>, ErrorBits =>)
   END_RUNG
   RUNG wire#powerrail
      { S7_Templates := "SrcType := Int" } NE_Contact(in1 := "MODE SELECTION DB"."DM FEED PUMP"."MODE BUFF", in2 := 1)
   END_RUNG wire#w1
   RUNG wire#powerrail
      I_Contact( "DI WATER TRANSFER DB"."P-502 AB/BC/CA" )
   END_RUNG wire#w1
   RUNG wire#powerrail
      Contact( "DI WATER TRANSFER DB"."P-502 AB/BC/CA" )
      wire#w2
      Move(in := 3, out1 => "PID_Compact_1".Mode)
   END_RUNG
   RUNG wire#w2
      Coil( "PID_Compact_1".ModeActivate )
   END_RUNG
   RUNG wire#powerrail
      { S7_Templates := "SrcType := Int" } NE_Contact(in1 := "MODE SELECTION DB"."DM FEED PUMP"."MODE BUFF", in2 := 1)
      wire#w3
      Move(in := 0, out1 => "PID_Compact_1".Mode)
   END_RUNG
   RUNG wire#powerrail
      I_Contact( "DI WATER TRANSFER DB"."P-502 AB/BC/CA" )
   END_RUNG wire#w3
   // the same network as SCL:
   "PID_Compact_1"(Reset := ("MODE SELECTION DB"."DM FEED PUMP"."MODE BUFF" <> 1) OR NOT "DI WATER TRANSFER DB"."P-502 AB/BC/CA",   // PID_Compact
                   Setpoint := "PID P-502 DB"."P-502"."IN SETPOINT",
                   Input := "PID P-502 DB"."P-502"."PV INPUT",
                   Output => "PID P-502 DB"."P-502"."P-502 MAIN NEWOUT");
   IF "DI WATER TRANSFER DB"."P-502 AB/BC/CA" THEN "PID_Compact_1".Mode := 3; END_IF;
   "PID_Compact_1".ModeActivate := "DI WATER TRANSFER DB"."P-502 AB/BC/CA";
   IF ("MODE SELECTION DB"."DM FEED PUMP"."MODE BUFF" <> 1) OR NOT "DI WATER TRANSFER DB"."P-502 AB/BC/CA" THEN
       "PID_Compact_1".Mode := 0;
   END_IF;
END_REGION

REGION Network 2: PID SET
   RUNG wire#powerrail
      Contact( "AlwaysTRUE" )
      wire#w1
      Move(in := "PID P-502 DB".PID_GAIN, out1 => "PID_Compact_1".Retain.CtrlParams.Gain)
   END_RUNG
   RUNG wire#w1
      Move(in := "PID P-502 DB".PID_I, out1 => "PID_Compact_1".Retain.CtrlParams.Ti)
   END_RUNG
   RUNG wire#w1
      Move(in := "PID P-502 DB".PID_D, out1 => "PID_Compact_1".Retain.CtrlParams.Td)
   END_RUNG
   // the same network as SCL:
   IF "AlwaysTRUE" THEN
       "PID_Compact_1".Retain.CtrlParams.Gain := "PID P-502 DB".PID_GAIN;
       "PID_Compact_1".Retain.CtrlParams.Ti := "PID P-502 DB".PID_I;
       "PID_Compact_1".Retain.CtrlParams.Td := "PID P-502 DB".PID_D;
   END_IF;
END_REGION
END_ORGANIZATION_BLOCK

DATA_BLOCK "SCALE AO_DB"   // DB126
// stored: InstanceOfName SCALE AO, InstanceOfType FB
"SCALE AO"
   // VAR_INPUT
   //    "SET RPM" : Real;
   //    "MIN RPM" : Real;
   //    "MAX RPM" : Real;
   //    "MIN RAW" : Int;
   //    "MAX RAW" : Int;
   // END_VAR
   // VAR_OUTPUT
   //    MODBUS : Int;
   // END_VAR
BEGIN
END_DATA_BLOCK

DATA_BLOCK "SCALE AO_DB_1"   // DB136
// stored: InstanceOfName SCALE AO, InstanceOfType FB
"SCALE AO"
   // VAR_INPUT
   //    "SET RPM" : Real;
   //    "MIN RPM" : Real;
   //    "MAX RPM" : Real;
   //    "MIN RAW" : Int;
   //    "MAX RAW" : Int;
   // END_VAR
   // VAR_OUTPUT
   //    MODBUS : Int;
   // END_VAR
BEGIN
END_DATA_BLOCK

DATA_BLOCK "SCALE AO_DB_2"   // DB149
// stored: InstanceOfName SCALE AO, InstanceOfType FB
"SCALE AO"
   // VAR_INPUT
   //    "SET RPM" : Real;
   //    "MIN RPM" : Real;
   //    "MAX RPM" : Real;
   //    "MIN RAW" : Int;
   //    "MAX RAW" : Int;
   // END_VAR
   // VAR_OUTPUT
   //    MODBUS : Int;
   // END_VAR
BEGIN
END_DATA_BLOCK

DATA_BLOCK "SCALE_DB"   // DB152
// stored: InstanceOfName SCALE, InstanceOfType FB
"SCALE"
   // VAR_INPUT
   //    "SCALE MIN" : Real;
   //    "SCALE MAX" : Real;
   //    INPUT : Int;
   //    "RAW MIN" : Int;
   //    "RAW MAX" : Int;
   // END_VAR
   // VAR_OUTPUT
   //    "PV VALUE" : Real;
   // END_VAR
BEGIN
END_DATA_BLOCK

DATA_BLOCK "SCALE_DB_1"   // DB155
// stored: InstanceOfName SCALE, InstanceOfType FB
"SCALE"
   // VAR_INPUT
   //    "SCALE MIN" : Real;
   //    "SCALE MAX" : Real;
   //    INPUT : Int;
   //    "RAW MIN" : Int;
   //    "RAW MAX" : Int;
   // END_VAR
   // VAR_OUTPUT
   //    "PV VALUE" : Real;
   // END_VAR
BEGIN
END_DATA_BLOCK

DATA_BLOCK "SCALE_DB_2"   // DB222
// stored: InstanceOfName SCALE, InstanceOfType FB
"SCALE"
   // VAR_INPUT
   //    "SCALE MIN" : Real;
   //    "SCALE MAX" : Real;
   //    INPUT : Int;
   //    "RAW MIN" : Int;
   //    "RAW MAX" : Int;
   // END_VAR
   // VAR_OUTPUT
   //    "PV VALUE" : Real;
   // END_VAR
BEGIN
END_DATA_BLOCK

DATA_BLOCK "SCALE_DB_3"   // DB213
// stored: InstanceOfName SCALE, InstanceOfType FB
"SCALE"
   // VAR_INPUT
   //    "SCALE MIN" : Real;
   //    "SCALE MAX" : Real;
   //    INPUT : Int;
   //    "RAW MIN" : Int;
   //    "RAW MAX" : Int;
   // END_VAR
   // VAR_OUTPUT
   //    "PV VALUE" : Real;
   // END_VAR
BEGIN
END_DATA_BLOCK

DATA_BLOCK "UV-601_SENSOR"   // DB227
// stored: InstanceOfName SCALE, InstanceOfType FB
"SCALE"
   // VAR_INPUT
   //    "SCALE MIN" : Real;
   //    "SCALE MAX" : Real;
   //    INPUT : Int;
   //    "RAW MIN" : Int;
   //    "RAW MAX" : Int;
   // END_VAR
   // VAR_OUTPUT
   //    "PV VALUE" : Real;
   // END_VAR
BEGIN
END_DATA_BLOCK

DATA_BLOCK "TIMING_MIN_DB"   // DB76
// stored: InstanceOfName TIMING_MIN, InstanceOfType FB
"TIMING_MIN"
BEGIN
END_DATA_BLOCK

DATA_BLOCK "TIMING_MIN_DB_1"   // DB82
// stored: InstanceOfName TIMING_MIN, InstanceOfType FB
"TIMING_MIN"
BEGIN
END_DATA_BLOCK

DATA_BLOCK "TIMING_MIN_DB_2"   // DB83
// stored: InstanceOfName TIMING_MIN, InstanceOfType FB
"TIMING_MIN"
BEGIN
END_DATA_BLOCK

DATA_BLOCK "TIMING_MIN_DB_3"   // DB156
// stored: InstanceOfName TIMING_MIN, InstanceOfType FB
"TIMING_MIN"
BEGIN
END_DATA_BLOCK

DATA_BLOCK "TIMING_MIN_DB_4"   // DB122
// stored: InstanceOfName TIMING_MIN, InstanceOfType FB
"TIMING_MIN"
BEGIN
END_DATA_BLOCK

DATA_BLOCK "TIMING_SECS_DB"   // DB108
// stored: InstanceOfName TIMING_SECS, InstanceOfType FB
"TIMING_SECS"
BEGIN
END_DATA_BLOCK

DATA_BLOCK "TIMING_SECS_DB_1"   // DB107
// stored: InstanceOfName TIMING_SECS, InstanceOfType FB
"TIMING_SECS"
BEGIN
END_DATA_BLOCK

DATA_BLOCK "TIMING_SECS_DB_10"   // DB128
// stored: InstanceOfName TIMING_SECS, InstanceOfType FB
"TIMING_SECS"
BEGIN
END_DATA_BLOCK

DATA_BLOCK "TIMING_SECS_DB_11"   // DB162
// stored: InstanceOfName TIMING_SECS, InstanceOfType FB
"TIMING_SECS"
BEGIN
END_DATA_BLOCK

DATA_BLOCK "TIMING_SECS_DB_12"   // DB131
// stored: InstanceOfName TIMING_SECS, InstanceOfType FB
"TIMING_SECS"
BEGIN
END_DATA_BLOCK

DATA_BLOCK "TIMING_SECS_DB_13"   // DB161
// stored: InstanceOfName TIMING_SECS, InstanceOfType FB
"TIMING_SECS"
BEGIN
END_DATA_BLOCK

DATA_BLOCK "TIMING_SECS_DB_14"   // DB160
// stored: InstanceOfName TIMING_SECS, InstanceOfType FB
"TIMING_SECS"
BEGIN
END_DATA_BLOCK

DATA_BLOCK "TIMING_SECS_DB_15"   // DB159
// stored: InstanceOfName TIMING_SECS, InstanceOfType FB
"TIMING_SECS"
BEGIN
END_DATA_BLOCK

DATA_BLOCK "TIMING_SECS_DB_16"   // DB157
// stored: InstanceOfName TIMING_SECS, InstanceOfType FB
"TIMING_SECS"
BEGIN
END_DATA_BLOCK

DATA_BLOCK "TIMING_SECS_DB_17"   // DB158
// stored: InstanceOfName TIMING_SECS, InstanceOfType FB
"TIMING_SECS"
BEGIN
END_DATA_BLOCK

DATA_BLOCK "TIMING_SECS_DB_2"   // DB106
// stored: InstanceOfName TIMING_SECS, InstanceOfType FB
"TIMING_SECS"
BEGIN
END_DATA_BLOCK

DATA_BLOCK "TIMING_SECS_DB_3"   // DB105
// stored: InstanceOfName TIMING_SECS, InstanceOfType FB
"TIMING_SECS"
BEGIN
END_DATA_BLOCK

DATA_BLOCK "TIMING_SECS_DB_4"   // DB90
// stored: InstanceOfName TIMING_SECS, InstanceOfType FB
"TIMING_SECS"
BEGIN
END_DATA_BLOCK

DATA_BLOCK "TIMING_SECS_DB_5"   // DB78
// stored: InstanceOfName TIMING_SECS, InstanceOfType FB
"TIMING_SECS"
BEGIN
END_DATA_BLOCK

DATA_BLOCK "TIMING_SECS_DB_6"   // DB112
// stored: InstanceOfName TIMING_SECS, InstanceOfType FB
"TIMING_SECS"
BEGIN
END_DATA_BLOCK

DATA_BLOCK "TIMING_SECS_DB_7"   // DB116
// stored: InstanceOfName TIMING_SECS, InstanceOfType FB
"TIMING_SECS"
BEGIN
END_DATA_BLOCK

DATA_BLOCK "TIMING_SECS_DB_8"   // DB119
// stored: InstanceOfName TIMING_SECS, InstanceOfType FB
"TIMING_SECS"
BEGIN
END_DATA_BLOCK

DATA_BLOCK "TIMING_SECS_DB_9"   // DB124
// stored: InstanceOfName TIMING_SECS, InstanceOfType FB
"TIMING_SECS"
BEGIN
END_DATA_BLOCK

DATA_BLOCK "TIMING_MIN_DB_6"   // DB211
// stored: InstanceOfName TIMING_MIN, InstanceOfType FB
"TIMING_MIN"
BEGIN
END_DATA_BLOCK

DATA_BLOCK "TIMING_SECS_DB_18"   // DB181
// stored: InstanceOfName TIMING_SECS, InstanceOfType FB
"TIMING_SECS"
BEGIN
END_DATA_BLOCK

DATA_BLOCK "CONDUCTIVITY INDICATOR CUM_TRANSMITTER-101"   // DB10
// stored: InstanceOfName SCALE, InstanceOfType FB
"SCALE"
   // VAR_INPUT
   //    "SCALE MIN" : Real;
   //    "SCALE MAX" : Real;
   //    INPUT : Int;
   //    "RAW MIN" : Int;
   //    "RAW MAX" : Int;
   // END_VAR
   // VAR_OUTPUT
   //    "PV VALUE" : Real;
   // END_VAR
BEGIN
END_DATA_BLOCK

DATA_BLOCK "DIFFRENTIAL PRESSURE TRANSMITTER-101_ANALOG"   // DB9
// stored: InstanceOfName SCALE, InstanceOfType FB
"SCALE"
   // VAR_INPUT
   //    "SCALE MIN" : Real;
   //    "SCALE MAX" : Real;
   //    INPUT : Int;
   //    "RAW MIN" : Int;
   //    "RAW MAX" : Int;
   // END_VAR
   // VAR_OUTPUT
   //    "PV VALUE" : Real;
   // END_VAR
BEGIN
END_DATA_BLOCK

DATA_BLOCK "DIFFRENTIAL PRESSURE_TRANSMITTER-201"   // DB11
// stored: InstanceOfName SCALE, InstanceOfType FB
"SCALE"
   // VAR_INPUT
   //    "SCALE MIN" : Real;
   //    "SCALE MAX" : Real;
   //    INPUT : Int;
   //    "RAW MIN" : Int;
   //    "RAW MAX" : Int;
   // END_VAR
   // VAR_OUTPUT
   //    "PV VALUE" : Real;
   // END_VAR
BEGIN
END_DATA_BLOCK

DATA_BLOCK "FLOW INDICATIOR TOTALISER_601"   // DB17
// stored: InstanceOfName SCALE, InstanceOfType FB
"SCALE"
   // VAR_INPUT
   //    "SCALE MIN" : Real;
   //    "SCALE MAX" : Real;
   //    INPUT : Int;
   //    "RAW MIN" : Int;
   //    "RAW MAX" : Int;
   // END_VAR
   // VAR_OUTPUT
   //    "PV VALUE" : Real;
   // END_VAR
BEGIN
END_DATA_BLOCK

DATA_BLOCK "FLOW INDICATIOR_TOTALISER-201"   // DB12
// stored: InstanceOfName SCALE, InstanceOfType FB
"SCALE"
   // VAR_INPUT
   //    "SCALE MIN" : Real;
   //    "SCALE MAX" : Real;
   //    INPUT : Int;
   //    "RAW MIN" : Int;
   //    "RAW MAX" : Int;
   // END_VAR
   // VAR_OUTPUT
   //    "PV VALUE" : Real;
   // END_VAR
BEGIN
END_DATA_BLOCK

DATA_BLOCK "LEVEL TRANSMITTER-101_ANALOG"   // DB6
// stored: InstanceOfName SCALE, InstanceOfType FB
"SCALE"
   // VAR_INPUT
   //    "SCALE MIN" : Real;
   //    "SCALE MAX" : Real;
   //    INPUT : Int;
   //    "RAW MIN" : Int;
   //    "RAW MAX" : Int;
   // END_VAR
   // VAR_OUTPUT
   //    "PV VALUE" : Real;
   // END_VAR
BEGIN
END_DATA_BLOCK

DATA_BLOCK "LEVEL TRANSMITTER-102_ANALOG"   // DB7
// stored: InstanceOfName SCALE, InstanceOfType FB
"SCALE"
   // VAR_INPUT
   //    "SCALE MIN" : Real;
   //    "SCALE MAX" : Real;
   //    INPUT : Int;
   //    "RAW MIN" : Int;
   //    "RAW MAX" : Int;
   // END_VAR
   // VAR_OUTPUT
   //    "PV VALUE" : Real;
   // END_VAR
BEGIN
END_DATA_BLOCK

DATA_BLOCK "LEVEL_TRANSMITTER-201"   // DB13
// stored: InstanceOfName SCALE, InstanceOfType FB
"SCALE"
   // VAR_INPUT
   //    "SCALE MIN" : Real;
   //    "SCALE MAX" : Real;
   //    INPUT : Int;
   //    "RAW MIN" : Int;
   //    "RAW MAX" : Int;
   // END_VAR
   // VAR_OUTPUT
   //    "PV VALUE" : Real;
   // END_VAR
BEGIN
END_DATA_BLOCK

DATA_BLOCK "LEVEL_TRANSMITTER-801"   // DB14
// stored: InstanceOfName SCALE, InstanceOfType FB
"SCALE"
   // VAR_INPUT
   //    "SCALE MIN" : Real;
   //    "SCALE MAX" : Real;
   //    INPUT : Int;
   //    "RAW MIN" : Int;
   //    "RAW MAX" : Int;
   // END_VAR
   // VAR_OUTPUT
   //    "PV VALUE" : Real;
   // END_VAR
BEGIN
END_DATA_BLOCK

DATA_BLOCK "PH INDICATOR CUM TRANSMITTER_601"   // DB18
// stored: InstanceOfName SCALE, InstanceOfType FB
"SCALE"
   // VAR_INPUT
   //    "SCALE MIN" : Real;
   //    "SCALE MAX" : Real;
   //    INPUT : Int;
   //    "RAW MIN" : Int;
   //    "RAW MAX" : Int;
   // END_VAR
   // VAR_OUTPUT
   //    "PV VALUE" : Real;
   // END_VAR
BEGIN
END_DATA_BLOCK

DATA_BLOCK "PRESSURE_TRANSMITTER 601"   // DB16
// stored: InstanceOfName SCALE, InstanceOfType FB
"SCALE"
   // VAR_INPUT
   //    "SCALE MIN" : Real;
   //    "SCALE MAX" : Real;
   //    INPUT : Int;
   //    "RAW MIN" : Int;
   //    "RAW MAX" : Int;
   // END_VAR
   // VAR_OUTPUT
   //    "PV VALUE" : Real;
   // END_VAR
BEGIN
END_DATA_BLOCK

DATA_BLOCK "RESISTIVITY CUM_TRANSMITTER 601"   // DB15
// stored: InstanceOfName SCALE, InstanceOfType FB
"SCALE"
   // VAR_INPUT
   //    "SCALE MIN" : Real;
   //    "SCALE MAX" : Real;
   //    INPUT : Int;
   //    "RAW MIN" : Int;
   //    "RAW MAX" : Int;
   // END_VAR
   // VAR_OUTPUT
   //    "PV VALUE" : Real;
   // END_VAR
BEGIN
END_DATA_BLOCK

DATA_BLOCK "ABFV 101 MULTIGRADE FILTER FULSH"   // DB44
// stored: InstanceOfName FLUSHING VALVE, InstanceOfType FB
"FLUSHING VALVE"
   // VAR_INPUT
   //    "SUBOUTPUT VALVE" : Bool;
   //    "OPEN FEEDBACK" : Bool;
   //    "CLOSE FEEDBACK" : Bool;
   // END_VAR
   // VAR_OUTPUT
   //    "OPEN OUTPUT VAVLE" : Bool;
   //    "CLOSE OUTPUT VAVLE" : Bool;
   // END_VAR
   // VAR
   //    TIMER_1 { S7_SetPoint := 'True'} : TON_TIME;
   //    "TIMER" { S7_SetPoint := 'True'} : TON_TIME;
   // END_VAR
BEGIN
END_DATA_BLOCK

DATA_BLOCK "ABFV 102 MULTIGRADE FILTER FLUSH"   // DB45
// stored: InstanceOfName FLUSHING VALVE, InstanceOfType FB
"FLUSHING VALVE"
   // VAR_INPUT
   //    "SUBOUTPUT VALVE" : Bool;
   //    "OPEN FEEDBACK" : Bool;
   //    "CLOSE FEEDBACK" : Bool;
   // END_VAR
   // VAR_OUTPUT
   //    "OPEN OUTPUT VAVLE" : Bool;
   //    "CLOSE OUTPUT VAVLE" : Bool;
   // END_VAR
   // VAR
   //    TIMER_1 { S7_SetPoint := 'True'} : TON_TIME;
   //    "TIMER" { S7_SetPoint := 'True'} : TON_TIME;
   // END_VAR
BEGIN
END_DATA_BLOCK

DATA_BLOCK "ABFV 103 MULTIGRADE FILTER FLUSH"   // DB46
// stored: InstanceOfName FLUSHING VALVE, InstanceOfType FB
"FLUSHING VALVE"
   // VAR_INPUT
   //    "SUBOUTPUT VALVE" : Bool;
   //    "OPEN FEEDBACK" : Bool;
   //    "CLOSE FEEDBACK" : Bool;
   // END_VAR
   // VAR_OUTPUT
   //    "OPEN OUTPUT VAVLE" : Bool;
   //    "CLOSE OUTPUT VAVLE" : Bool;
   // END_VAR
   // VAR
   //    TIMER_1 { S7_SetPoint := 'True'} : TON_TIME;
   //    "TIMER" { S7_SetPoint := 'True'} : TON_TIME;
   // END_VAR
BEGIN
END_DATA_BLOCK

DATA_BLOCK "ABFV 104 MULTIGRADE FILTER FLUSH"   // DB47
// stored: InstanceOfName FLUSHING VALVE, InstanceOfType FB
"FLUSHING VALVE"
   // VAR_INPUT
   //    "SUBOUTPUT VALVE" : Bool;
   //    "OPEN FEEDBACK" : Bool;
   //    "CLOSE FEEDBACK" : Bool;
   // END_VAR
   // VAR_OUTPUT
   //    "OPEN OUTPUT VAVLE" : Bool;
   //    "CLOSE OUTPUT VAVLE" : Bool;
   // END_VAR
   // VAR
   //    TIMER_1 { S7_SetPoint := 'True'} : TON_TIME;
   //    "TIMER" { S7_SetPoint := 'True'} : TON_TIME;
   // END_VAR
BEGIN
END_DATA_BLOCK

DATA_BLOCK "ABFV 105 MULTIGRADE FILTER FLUSH"   // DB48
// stored: InstanceOfName FLUSHING VALVE, InstanceOfType FB
"FLUSHING VALVE"
   // VAR_INPUT
   //    "SUBOUTPUT VALVE" : Bool;
   //    "OPEN FEEDBACK" : Bool;
   //    "CLOSE FEEDBACK" : Bool;
   // END_VAR
   // VAR_OUTPUT
   //    "OPEN OUTPUT VAVLE" : Bool;
   //    "CLOSE OUTPUT VAVLE" : Bool;
   // END_VAR
   // VAR
   //    TIMER_1 { S7_SetPoint := 'True'} : TON_TIME;
   //    "TIMER" { S7_SetPoint := 'True'} : TON_TIME;
   // END_VAR
BEGIN
END_DATA_BLOCK

DATA_BLOCK "ABFV 201 FEED BACK FLUSH"   // DB175
// stored: InstanceOfName FLUSHING VALVE, InstanceOfType FB
"FLUSHING VALVE"
   // VAR_INPUT
   //    "SUBOUTPUT VALVE" : Bool;
   //    "OPEN FEEDBACK" : Bool;
   //    "CLOSE FEEDBACK" : Bool;
   // END_VAR
   // VAR_OUTPUT
   //    "OPEN OUTPUT VAVLE" : Bool;
   //    "CLOSE OUTPUT VAVLE" : Bool;
   // END_VAR
   // VAR
   //    TIMER_1 { S7_SetPoint := 'True'} : TON_TIME;
   //    "TIMER" { S7_SetPoint := 'True'} : TON_TIME;
   // END_VAR
BEGIN
END_DATA_BLOCK

DATA_BLOCK "ABFV 202 FEED BACK FLUSH"   // DB50
// stored: InstanceOfName FLUSHING VALVE, InstanceOfType FB
"FLUSHING VALVE"
   // VAR_INPUT
   //    "SUBOUTPUT VALVE" : Bool;
   //    "OPEN FEEDBACK" : Bool;
   //    "CLOSE FEEDBACK" : Bool;
   // END_VAR
   // VAR_OUTPUT
   //    "OPEN OUTPUT VAVLE" : Bool;
   //    "CLOSE OUTPUT VAVLE" : Bool;
   // END_VAR
   // VAR
   //    TIMER_1 { S7_SetPoint := 'True'} : TON_TIME;
   //    "TIMER" { S7_SetPoint := 'True'} : TON_TIME;
   // END_VAR
BEGIN
END_DATA_BLOCK

DATA_BLOCK "ABFV 203 FEED BACK FLUSH"   // DB51
// stored: InstanceOfName FLUSHING VALVE, InstanceOfType FB
"FLUSHING VALVE"
   // VAR_INPUT
   //    "SUBOUTPUT VALVE" : Bool;
   //    "OPEN FEEDBACK" : Bool;
   //    "CLOSE FEEDBACK" : Bool;
   // END_VAR
   // VAR_OUTPUT
   //    "OPEN OUTPUT VAVLE" : Bool;
   //    "CLOSE OUTPUT VAVLE" : Bool;
   // END_VAR
   // VAR
   //    TIMER_1 { S7_SetPoint := 'True'} : TON_TIME;
   //    "TIMER" { S7_SetPoint := 'True'} : TON_TIME;
   // END_VAR
BEGIN
END_DATA_BLOCK

DATA_BLOCK "ABFV 204 FEED BACK FLUSH"   // DB52
// stored: InstanceOfName FLUSHING VALVE, InstanceOfType FB
"FLUSHING VALVE"
   // VAR_INPUT
   //    "SUBOUTPUT VALVE" : Bool;
   //    "OPEN FEEDBACK" : Bool;
   //    "CLOSE FEEDBACK" : Bool;
   // END_VAR
   // VAR_OUTPUT
   //    "OPEN OUTPUT VAVLE" : Bool;
   //    "CLOSE OUTPUT VAVLE" : Bool;
   // END_VAR
   // VAR
   //    TIMER_1 { S7_SetPoint := 'True'} : TON_TIME;
   //    "TIMER" { S7_SetPoint := 'True'} : TON_TIME;
   // END_VAR
BEGIN
END_DATA_BLOCK

DATA_BLOCK "ABFV 205 FEED BACK FLUSH"   // DB53
// stored: InstanceOfName FLUSHING VALVE, InstanceOfType FB
"FLUSHING VALVE"
   // VAR_INPUT
   //    "SUBOUTPUT VALVE" : Bool;
   //    "OPEN FEEDBACK" : Bool;
   //    "CLOSE FEEDBACK" : Bool;
   // END_VAR
   // VAR_OUTPUT
   //    "OPEN OUTPUT VAVLE" : Bool;
   //    "CLOSE OUTPUT VAVLE" : Bool;
   // END_VAR
   // VAR
   //    TIMER_1 { S7_SetPoint := 'True'} : TON_TIME;
   //    "TIMER" { S7_SetPoint := 'True'} : TON_TIME;
   // END_VAR
BEGIN
END_DATA_BLOCK

DATA_BLOCK "ABFV 206 FEED BACK FLUSH"   // DB54
// stored: InstanceOfName FLUSHING VALVE, InstanceOfType FB
"FLUSHING VALVE"
   // VAR_INPUT
   //    "SUBOUTPUT VALVE" : Bool;
   //    "OPEN FEEDBACK" : Bool;
   //    "CLOSE FEEDBACK" : Bool;
   // END_VAR
   // VAR_OUTPUT
   //    "OPEN OUTPUT VAVLE" : Bool;
   //    "CLOSE OUTPUT VAVLE" : Bool;
   // END_VAR
   // VAR
   //    TIMER_1 { S7_SetPoint := 'True'} : TON_TIME;
   //    "TIMER" { S7_SetPoint := 'True'} : TON_TIME;
   // END_VAR
BEGIN
END_DATA_BLOCK

DATA_BLOCK "ABFV 207 FEED BACK FLUSH"   // DB55
// stored: InstanceOfName FLUSHING VALVE, InstanceOfType FB
"FLUSHING VALVE"
   // VAR_INPUT
   //    "SUBOUTPUT VALVE" : Bool;
   //    "OPEN FEEDBACK" : Bool;
   //    "CLOSE FEEDBACK" : Bool;
   // END_VAR
   // VAR_OUTPUT
   //    "OPEN OUTPUT VAVLE" : Bool;
   //    "CLOSE OUTPUT VAVLE" : Bool;
   // END_VAR
   // VAR
   //    TIMER_1 { S7_SetPoint := 'True'} : TON_TIME;
   //    "TIMER" { S7_SetPoint := 'True'} : TON_TIME;
   // END_VAR
BEGIN
END_DATA_BLOCK

DATA_BLOCK "ABFV 208 FEED BACK FLUSH"   // DB56
// stored: InstanceOfName FLUSHING VALVE, InstanceOfType FB
"FLUSHING VALVE"
   // VAR_INPUT
   //    "SUBOUTPUT VALVE" : Bool;
   //    "OPEN FEEDBACK" : Bool;
   //    "CLOSE FEEDBACK" : Bool;
   // END_VAR
   // VAR_OUTPUT
   //    "OPEN OUTPUT VAVLE" : Bool;
   //    "CLOSE OUTPUT VAVLE" : Bool;
   // END_VAR
   // VAR
   //    TIMER_1 { S7_SetPoint := 'True'} : TON_TIME;
   //    "TIMER" { S7_SetPoint := 'True'} : TON_TIME;
   // END_VAR
BEGIN
END_DATA_BLOCK

DATA_BLOCK "ABFV-501 FULSE"   // DB42
// stored: InstanceOfName FLUSHING VALVE, InstanceOfType FB
"FLUSHING VALVE"
   // VAR_INPUT
   //    "SUBOUTPUT VALVE" : Bool;
   //    "OPEN FEEDBACK" : Bool;
   //    "CLOSE FEEDBACK" : Bool;
   // END_VAR
   // VAR_OUTPUT
   //    "OPEN OUTPUT VAVLE" : Bool;
   //    "CLOSE OUTPUT VAVLE" : Bool;
   // END_VAR
   // VAR
   //    TIMER_1 { S7_SetPoint := 'True'} : TON_TIME;
   //    "TIMER" { S7_SetPoint := 'True'} : TON_TIME;
   // END_VAR
BEGIN
END_DATA_BLOCK

DATA_BLOCK "ABFV-502 FULSE"   // DB43
// stored: InstanceOfName FLUSHING VALVE, InstanceOfType FB
"FLUSHING VALVE"
   // VAR_INPUT
   //    "SUBOUTPUT VALVE" : Bool;
   //    "OPEN FEEDBACK" : Bool;
   //    "CLOSE FEEDBACK" : Bool;
   // END_VAR
   // VAR_OUTPUT
   //    "OPEN OUTPUT VAVLE" : Bool;
   //    "CLOSE OUTPUT VAVLE" : Bool;
   // END_VAR
   // VAR
   //    TIMER_1 { S7_SetPoint := 'True'} : TON_TIME;
   //    "TIMER" { S7_SetPoint := 'True'} : TON_TIME;
   // END_VAR
BEGIN
END_DATA_BLOCK

DATA_BLOCK "ABV 201 FEED BACK FLUSH"   // DB49
// stored: InstanceOfName FLUSHING VALVE, InstanceOfType FB
"FLUSHING VALVE"
   // VAR_INPUT
   //    "SUBOUTPUT VALVE" : Bool;
   //    "OPEN FEEDBACK" : Bool;
   //    "CLOSE FEEDBACK" : Bool;
   // END_VAR
   // VAR_OUTPUT
   //    "OPEN OUTPUT VAVLE" : Bool;
   //    "CLOSE OUTPUT VAVLE" : Bool;
   // END_VAR
   // VAR
   //    TIMER_1 { S7_SetPoint := 'True'} : TON_TIME;
   //    "TIMER" { S7_SetPoint := 'True'} : TON_TIME;
   // END_VAR
BEGIN
END_DATA_BLOCK

DATA_BLOCK "TIMING_MIN_DB_5"   // DB190
// stored: InstanceOfName TIMING_MIN, InstanceOfType FB
"TIMING_MIN"
BEGIN
END_DATA_BLOCK

DATA_BLOCK "GET_DB"   // DB166
// stored: InstanceOfName GET_SFB, OfSystemLibElement GET, OfSystemLibVersion 1.3
"GET_SFB"
   // VAR_INPUT
   //    REQ : Bool;
   //    ID : Word;
   // END_VAR
   // VAR_OUTPUT
   //    NDR : Bool;
   //    ERROR : Bool;
   //    STATUS : Word;
   // END_VAR
   // VAR_IN_OUT
   //    ADDR_1 : Remote;
   //    ADDR_2 : Remote;
   //    ADDR_3 : Remote;
   //    ADDR_4 : Remote;
   //    RD_1 : Variant;
   //    RD_2 : Variant;
   //    RD_3 : Variant;
   //    RD_4 : Variant;
   // END_VAR
BEGIN
END_DATA_BLOCK

DATA_BLOCK "IEC_Counter_0_DB"   // DB163
{ S7_Optimized_Access := 'TRUE' }
// stored: InstanceOfName IEC_COUNTER, OfSystemLibElement IEC_COUNTER, OfSystemLibVersion 1.0
"IEC_COUNTER"
   // VAR RETAIN
   //    CU : Bool;
   //    CD : Bool;
   //    R : Bool;
   //    LD : Bool;
   //    QU : Bool;
   //    QD : Bool;
   //    PV : Int;
   //    CV : Int;
   // END_VAR
BEGIN
END_DATA_BLOCK

DATA_BLOCK "IEC_Counter_0_DB_1"   // DB224
{ S7_Optimized_Access := 'TRUE' }
// stored: InstanceOfName IEC_COUNTER, OfSystemLibElement IEC_COUNTER, OfSystemLibVersion 1.0
"IEC_COUNTER"
   // VAR RETAIN
   //    CU : Bool;
   //    CD : Bool;
   //    R : Bool;
   //    LD : Bool;
   //    QU : Bool;
   //    QD : Bool;
   //    PV : Int;
   //    CV : Int;
   // END_VAR
BEGIN
END_DATA_BLOCK

DATA_BLOCK "IEC_Timer_0_DB"   // DB22
{ S7_Optimized_Access := 'TRUE' }
// stored: InstanceOfName IEC_TIMER, OfSystemLibElement IEC_TIMER, OfSystemLibVersion 1.0
"IEC_TIMER"
   // VAR
   //    PT : Time;
   //    ET { ExternalWritable := 'False'} : Time;
   //    IN : Bool;
   //    Q { ExternalWritable := 'False'} : Bool;
   // END_VAR
BEGIN
END_DATA_BLOCK

DATA_BLOCK "IEC_Timer_0_DB_1"   // DB23
{ S7_Optimized_Access := 'TRUE' }
// stored: InstanceOfName IEC_TIMER, OfSystemLibElement IEC_TIMER, OfSystemLibVersion 1.0
"IEC_TIMER"
   // VAR
   //    PT : Time;
   //    ET { ExternalWritable := 'False'} : Time;
   //    IN : Bool;
   //    Q { ExternalWritable := 'False'} : Bool;
   // END_VAR
BEGIN
END_DATA_BLOCK

DATA_BLOCK "IEC_Timer_0_DB_10"   // DB32
{ S7_Optimized_Access := 'TRUE' }
// stored: InstanceOfName IEC_TIMER, OfSystemLibElement IEC_TIMER, OfSystemLibVersion 1.0
"IEC_TIMER"
   // VAR
   //    PT : Time;
   //    ET { ExternalWritable := 'False'} : Time;
   //    IN : Bool;
   //    Q { ExternalWritable := 'False'} : Bool;
   // END_VAR
BEGIN
END_DATA_BLOCK

DATA_BLOCK "IEC_Timer_0_DB_100"   // DB207
{ S7_Optimized_Access := 'TRUE' }
// stored: InstanceOfName IEC_TIMER, OfSystemLibElement IEC_TIMER, OfSystemLibVersion 1.0
"IEC_TIMER"
   // VAR
   //    PT : Time;
   //    ET { ExternalWritable := 'False'} : Time;
   //    IN : Bool;
   //    Q { ExternalWritable := 'False'} : Bool;
   // END_VAR
BEGIN
END_DATA_BLOCK

DATA_BLOCK "IEC_Timer_0_DB_101"   // DB178
{ S7_Optimized_Access := 'TRUE' }
// stored: InstanceOfName IEC_TIMER, OfSystemLibElement IEC_TIMER, OfSystemLibVersion 1.0
"IEC_TIMER"
   // VAR
   //    PT : Time;
   //    ET { ExternalWritable := 'False'} : Time;
   //    IN : Bool;
   //    Q { ExternalWritable := 'False'} : Bool;
   // END_VAR
BEGIN
END_DATA_BLOCK

DATA_BLOCK "IEC_Timer_0_DB_102"   // DB219
{ S7_Optimized_Access := 'TRUE' }
// stored: InstanceOfName IEC_TIMER, OfSystemLibElement IEC_TIMER, OfSystemLibVersion 1.0
"IEC_TIMER"
   // VAR
   //    PT : Time;
   //    ET { ExternalWritable := 'False'} : Time;
   //    IN : Bool;
   //    Q { ExternalWritable := 'False'} : Bool;
   // END_VAR
BEGIN
END_DATA_BLOCK

DATA_BLOCK "IEC_Timer_0_DB_103"   // DB180
{ S7_Optimized_Access := 'TRUE' }
// stored: InstanceOfName IEC_TIMER, OfSystemLibElement IEC_TIMER, OfSystemLibVersion 1.0
"IEC_TIMER"
   // VAR
   //    PT : Time;
   //    ET { ExternalWritable := 'False'} : Time;
   //    IN : Bool;
   //    Q { ExternalWritable := 'False'} : Bool;
   // END_VAR
BEGIN
END_DATA_BLOCK

DATA_BLOCK "IEC_Timer_0_DB_104"   // DB182
{ S7_Optimized_Access := 'TRUE' }
// stored: InstanceOfName IEC_TIMER, OfSystemLibElement IEC_TIMER, OfSystemLibVersion 1.0
"IEC_TIMER"
   // VAR
   //    PT : Time;
   //    ET { ExternalWritable := 'False'} : Time;
   //    IN : Bool;
   //    Q { ExternalWritable := 'False'} : Bool;
   // END_VAR
BEGIN
END_DATA_BLOCK

DATA_BLOCK "IEC_Timer_0_DB_105"   // DB183
{ S7_Optimized_Access := 'TRUE' }
// stored: InstanceOfName IEC_TIMER, OfSystemLibElement IEC_TIMER, OfSystemLibVersion 1.0
"IEC_TIMER"
   // VAR
   //    PT : Time;
   //    ET { ExternalWritable := 'False'} : Time;
   //    IN : Bool;
   //    Q { ExternalWritable := 'False'} : Bool;
   // END_VAR
BEGIN
END_DATA_BLOCK

DATA_BLOCK "IEC_Timer_0_DB_106"   // DB184
{ S7_Optimized_Access := 'TRUE' }
// stored: InstanceOfName IEC_TIMER, OfSystemLibElement IEC_TIMER, OfSystemLibVersion 1.0
"IEC_TIMER"
   // VAR
   //    PT : Time;
   //    ET { ExternalWritable := 'False'} : Time;
   //    IN : Bool;
   //    Q { ExternalWritable := 'False'} : Bool;
   // END_VAR
BEGIN
END_DATA_BLOCK

DATA_BLOCK "IEC_Timer_0_DB_107"   // DB185
{ S7_Optimized_Access := 'TRUE' }
// stored: InstanceOfName IEC_TIMER, OfSystemLibElement IEC_TIMER, OfSystemLibVersion 1.0
"IEC_TIMER"
   // VAR
   //    PT : Time;
   //    ET { ExternalWritable := 'False'} : Time;
   //    IN : Bool;
   //    Q { ExternalWritable := 'False'} : Bool;
   // END_VAR
BEGIN
END_DATA_BLOCK

DATA_BLOCK "IEC_Timer_0_DB_108"   // DB186
{ S7_Optimized_Access := 'TRUE' }
// stored: InstanceOfName IEC_TIMER, OfSystemLibElement IEC_TIMER, OfSystemLibVersion 1.0
"IEC_TIMER"
   // VAR
   //    PT : Time;
   //    ET { ExternalWritable := 'False'} : Time;
   //    IN : Bool;
   //    Q { ExternalWritable := 'False'} : Bool;
   // END_VAR
BEGIN
END_DATA_BLOCK

DATA_BLOCK "IEC_Timer_0_DB_109"   // DB187
{ S7_Optimized_Access := 'TRUE' }
// stored: InstanceOfName IEC_TIMER, OfSystemLibElement IEC_TIMER, OfSystemLibVersion 1.0
"IEC_TIMER"
   // VAR
   //    PT : Time;
   //    ET { ExternalWritable := 'False'} : Time;
   //    IN : Bool;
   //    Q { ExternalWritable := 'False'} : Bool;
   // END_VAR
BEGIN
END_DATA_BLOCK

DATA_BLOCK "IEC_Timer_0_DB_11"   // DB33
{ S7_Optimized_Access := 'TRUE' }
// stored: InstanceOfName IEC_TIMER, OfSystemLibElement IEC_TIMER, OfSystemLibVersion 1.0
"IEC_TIMER"
   // VAR
   //    PT : Time;
   //    ET { ExternalWritable := 'False'} : Time;
   //    IN : Bool;
   //    Q { ExternalWritable := 'False'} : Bool;
   // END_VAR
BEGIN
END_DATA_BLOCK

DATA_BLOCK "IEC_Timer_0_DB_110"   // DB188
{ S7_Optimized_Access := 'TRUE' }
// stored: InstanceOfName IEC_TIMER, OfSystemLibElement IEC_TIMER, OfSystemLibVersion 1.0
"IEC_TIMER"
   // VAR
   //    PT : Time;
   //    ET { ExternalWritable := 'False'} : Time;
   //    IN : Bool;
   //    Q { ExternalWritable := 'False'} : Bool;
   // END_VAR
BEGIN
END_DATA_BLOCK

DATA_BLOCK "IEC_Timer_0_DB_111"   // DB189
{ S7_Optimized_Access := 'TRUE' }
// stored: InstanceOfName IEC_TIMER, OfSystemLibElement IEC_TIMER, OfSystemLibVersion 1.0
"IEC_TIMER"
   // VAR
   //    PT : Time;
   //    ET { ExternalWritable := 'False'} : Time;
   //    IN : Bool;
   //    Q { ExternalWritable := 'False'} : Bool;
   // END_VAR
BEGIN
END_DATA_BLOCK

DATA_BLOCK "IEC_Timer_0_DB_112"   // DB191
{ S7_Optimized_Access := 'TRUE' }
// stored: InstanceOfName IEC_TIMER, OfSystemLibElement IEC_TIMER, OfSystemLibVersion 1.0
"IEC_TIMER"
   // VAR
   //    PT : Time;
   //    ET { ExternalWritable := 'False'} : Time;
   //    IN : Bool;
   //    Q { ExternalWritable := 'False'} : Bool;
   // END_VAR
BEGIN
END_DATA_BLOCK

DATA_BLOCK "IEC_Timer_0_DB_113"   // DB192
{ S7_Optimized_Access := 'TRUE' }
// stored: InstanceOfName IEC_TIMER, OfSystemLibElement IEC_TIMER, OfSystemLibVersion 1.0
"IEC_TIMER"
   // VAR
   //    PT : Time;
   //    ET { ExternalWritable := 'False'} : Time;
   //    IN : Bool;
   //    Q { ExternalWritable := 'False'} : Bool;
   // END_VAR
BEGIN
END_DATA_BLOCK

DATA_BLOCK "IEC_Timer_0_DB_114"   // DB226
{ S7_Optimized_Access := 'TRUE' }
// stored: InstanceOfName IEC_TIMER, OfSystemLibElement IEC_TIMER, OfSystemLibVersion 1.0
"IEC_TIMER"
   // VAR
   //    PT : Time;
   //    ET { ExternalWritable := 'False'} : Time;
   //    IN : Bool;
   //    Q { ExternalWritable := 'False'} : Bool;
   // END_VAR
BEGIN
END_DATA_BLOCK

DATA_BLOCK "IEC_Timer_0_DB_115"   // DB229
{ S7_Optimized_Access := 'TRUE' }
// stored: InstanceOfName IEC_TIMER, OfSystemLibElement IEC_TIMER, OfSystemLibVersion 1.0
"IEC_TIMER"
   // VAR
   //    PT : Time;
   //    ET { ExternalWritable := 'False'} : Time;
   //    IN : Bool;
   //    Q { ExternalWritable := 'False'} : Bool;
   // END_VAR
BEGIN
END_DATA_BLOCK

DATA_BLOCK "IEC_Timer_0_DB_116"   // DB231
{ S7_Optimized_Access := 'TRUE' }
// stored: InstanceOfName IEC_TIMER, OfSystemLibElement IEC_TIMER, OfSystemLibVersion 1.0
"IEC_TIMER"
   // VAR
   //    PT : Time;
   //    ET { ExternalWritable := 'False'} : Time;
   //    IN : Bool;
   //    Q { ExternalWritable := 'False'} : Bool;
   // END_VAR
BEGIN
END_DATA_BLOCK

DATA_BLOCK "IEC_Timer_0_DB_117"   // DB232
{ S7_Optimized_Access := 'TRUE' }
// stored: InstanceOfName IEC_TIMER, OfSystemLibElement IEC_TIMER, OfSystemLibVersion 1.0
"IEC_TIMER"
   // VAR
   //    PT : Time;
   //    ET { ExternalWritable := 'False'} : Time;
   //    IN : Bool;
   //    Q { ExternalWritable := 'False'} : Bool;
   // END_VAR
BEGIN
END_DATA_BLOCK

DATA_BLOCK "IEC_Timer_0_DB_118"   // DB177
{ S7_Optimized_Access := 'TRUE' }
// stored: InstanceOfName IEC_TIMER, OfSystemLibElement IEC_TIMER, OfSystemLibVersion 1.0
"IEC_TIMER"
   // VAR
   //    PT : Time;
   //    ET { ExternalWritable := 'False'} : Time;
   //    IN : Bool;
   //    Q { ExternalWritable := 'False'} : Bool;
   // END_VAR
BEGIN
END_DATA_BLOCK

DATA_BLOCK "IEC_Timer_0_DB_119"   // DB179
{ S7_Optimized_Access := 'TRUE' }
// stored: InstanceOfName IEC_TIMER, OfSystemLibElement IEC_TIMER, OfSystemLibVersion 1.0
"IEC_TIMER"
   // VAR
   //    PT : Time;
   //    ET { ExternalWritable := 'False'} : Time;
   //    IN : Bool;
   //    Q { ExternalWritable := 'False'} : Bool;
   // END_VAR
BEGIN
END_DATA_BLOCK

DATA_BLOCK "IEC_Timer_0_DB_12"   // DB34
{ S7_Optimized_Access := 'TRUE' }
// stored: InstanceOfName IEC_TIMER, OfSystemLibElement IEC_TIMER, OfSystemLibVersion 1.0
"IEC_TIMER"
   // VAR
   //    PT : Time;
   //    ET { ExternalWritable := 'False'} : Time;
   //    IN : Bool;
   //    Q { ExternalWritable := 'False'} : Bool;
   // END_VAR
BEGIN
END_DATA_BLOCK

DATA_BLOCK "IEC_Timer_0_DB_120"   // DB193
{ S7_Optimized_Access := 'TRUE' }
// stored: InstanceOfName IEC_TIMER, OfSystemLibElement IEC_TIMER, OfSystemLibVersion 1.0
"IEC_TIMER"
   // VAR
   //    PT : Time;
   //    ET { ExternalWritable := 'False'} : Time;
   //    IN : Bool;
   //    Q { ExternalWritable := 'False'} : Bool;
   // END_VAR
BEGIN
END_DATA_BLOCK

DATA_BLOCK "IEC_Timer_0_DB_121"   // DB194
{ S7_Optimized_Access := 'TRUE' }
// stored: InstanceOfName IEC_TIMER, OfSystemLibElement IEC_TIMER, OfSystemLibVersion 1.0
"IEC_TIMER"
   // VAR
   //    PT : Time;
   //    ET { ExternalWritable := 'False'} : Time;
   //    IN : Bool;
   //    Q { ExternalWritable := 'False'} : Bool;
   // END_VAR
BEGIN
END_DATA_BLOCK

DATA_BLOCK "IEC_Timer_0_DB_122"   // DB195
{ S7_Optimized_Access := 'TRUE' }
// stored: InstanceOfName IEC_TIMER, OfSystemLibElement IEC_TIMER, OfSystemLibVersion 1.0
"IEC_TIMER"
   // VAR
   //    PT : Time;
   //    ET { ExternalWritable := 'False'} : Time;
   //    IN : Bool;
   //    Q { ExternalWritable := 'False'} : Bool;
   // END_VAR
BEGIN
END_DATA_BLOCK

DATA_BLOCK "IEC_Timer_0_DB_123"   // DB196
{ S7_Optimized_Access := 'TRUE' }
// stored: InstanceOfName IEC_TIMER, OfSystemLibElement IEC_TIMER, OfSystemLibVersion 1.0
"IEC_TIMER"
   // VAR
   //    PT : Time;
   //    ET { ExternalWritable := 'False'} : Time;
   //    IN : Bool;
   //    Q { ExternalWritable := 'False'} : Bool;
   // END_VAR
BEGIN
END_DATA_BLOCK

DATA_BLOCK "IEC_Timer_0_DB_124"   // DB197
{ S7_Optimized_Access := 'TRUE' }
// stored: InstanceOfName IEC_TIMER, OfSystemLibElement IEC_TIMER, OfSystemLibVersion 1.0
"IEC_TIMER"
   // VAR
   //    PT : Time;
   //    ET { ExternalWritable := 'False'} : Time;
   //    IN : Bool;
   //    Q { ExternalWritable := 'False'} : Bool;
   // END_VAR
BEGIN
END_DATA_BLOCK

DATA_BLOCK "IEC_Timer_0_DB_125"   // DB198
{ S7_Optimized_Access := 'TRUE' }
// stored: InstanceOfName IEC_TIMER, OfSystemLibElement IEC_TIMER, OfSystemLibVersion 1.0
"IEC_TIMER"
   // VAR
   //    PT : Time;
   //    ET { ExternalWritable := 'False'} : Time;
   //    IN : Bool;
   //    Q { ExternalWritable := 'False'} : Bool;
   // END_VAR
BEGIN
END_DATA_BLOCK

DATA_BLOCK "IEC_Timer_0_DB_126"   // DB199
{ S7_Optimized_Access := 'TRUE' }
// stored: InstanceOfName IEC_TIMER, OfSystemLibElement IEC_TIMER, OfSystemLibVersion 1.0
"IEC_TIMER"
   // VAR
   //    PT : Time;
   //    ET { ExternalWritable := 'False'} : Time;
   //    IN : Bool;
   //    Q { ExternalWritable := 'False'} : Bool;
   // END_VAR
BEGIN
END_DATA_BLOCK

DATA_BLOCK "IEC_Timer_0_DB_127"   // DB200
{ S7_Optimized_Access := 'TRUE' }
// stored: InstanceOfName IEC_TIMER, OfSystemLibElement IEC_TIMER, OfSystemLibVersion 1.0
"IEC_TIMER"
   // VAR
   //    PT : Time;
   //    ET { ExternalWritable := 'False'} : Time;
   //    IN : Bool;
   //    Q { ExternalWritable := 'False'} : Bool;
   // END_VAR
BEGIN
END_DATA_BLOCK

DATA_BLOCK "IEC_Timer_0_DB_128"   // DB201
{ S7_Optimized_Access := 'TRUE' }
// stored: InstanceOfName IEC_TIMER, OfSystemLibElement IEC_TIMER, OfSystemLibVersion 1.0
"IEC_TIMER"
   // VAR
   //    PT : Time;
   //    ET { ExternalWritable := 'False'} : Time;
   //    IN : Bool;
   //    Q { ExternalWritable := 'False'} : Bool;
   // END_VAR
BEGIN
END_DATA_BLOCK

DATA_BLOCK "IEC_Timer_0_DB_129"   // DB202
{ S7_Optimized_Access := 'TRUE' }
// stored: InstanceOfName IEC_TIMER, OfSystemLibElement IEC_TIMER, OfSystemLibVersion 1.0
"IEC_TIMER"
   // VAR
   //    PT : Time;
   //    ET { ExternalWritable := 'False'} : Time;
   //    IN : Bool;
   //    Q { ExternalWritable := 'False'} : Bool;
   // END_VAR
BEGIN
END_DATA_BLOCK

DATA_BLOCK "IEC_Timer_0_DB_13"   // DB35
{ S7_Optimized_Access := 'TRUE' }
// stored: InstanceOfName IEC_TIMER, OfSystemLibElement IEC_TIMER, OfSystemLibVersion 1.0
"IEC_TIMER"
   // VAR
   //    PT : Time;
   //    ET { ExternalWritable := 'False'} : Time;
   //    IN : Bool;
   //    Q { ExternalWritable := 'False'} : Bool;
   // END_VAR
BEGIN
END_DATA_BLOCK

DATA_BLOCK "IEC_Timer_0_DB_130"   // DB203
{ S7_Optimized_Access := 'TRUE' }
// stored: InstanceOfName IEC_TIMER, OfSystemLibElement IEC_TIMER, OfSystemLibVersion 1.0
"IEC_TIMER"
   // VAR
   //    PT : Time;
   //    ET { ExternalWritable := 'False'} : Time;
   //    IN : Bool;
   //    Q { ExternalWritable := 'False'} : Bool;
   // END_VAR
BEGIN
END_DATA_BLOCK

DATA_BLOCK "IEC_Timer_0_DB_131"   // DB204
{ S7_Optimized_Access := 'TRUE' }
// stored: InstanceOfName IEC_TIMER, OfSystemLibElement IEC_TIMER, OfSystemLibVersion 1.0
"IEC_TIMER"
   // VAR
   //    PT : Time;
   //    ET { ExternalWritable := 'False'} : Time;
   //    IN : Bool;
   //    Q { ExternalWritable := 'False'} : Bool;
   // END_VAR
BEGIN
END_DATA_BLOCK

DATA_BLOCK "IEC_Timer_0_DB_132"   // DB205
{ S7_Optimized_Access := 'TRUE' }
// stored: InstanceOfName IEC_TIMER, OfSystemLibElement IEC_TIMER, OfSystemLibVersion 1.0
"IEC_TIMER"
   // VAR
   //    PT : Time;
   //    ET { ExternalWritable := 'False'} : Time;
   //    IN : Bool;
   //    Q { ExternalWritable := 'False'} : Bool;
   // END_VAR
BEGIN
END_DATA_BLOCK

DATA_BLOCK "IEC_Timer_0_DB_133"   // DB206
{ S7_Optimized_Access := 'TRUE' }
// stored: InstanceOfName IEC_TIMER, OfSystemLibElement IEC_TIMER, OfSystemLibVersion 1.0
"IEC_TIMER"
   // VAR
   //    PT : Time;
   //    ET { ExternalWritable := 'False'} : Time;
   //    IN : Bool;
   //    Q { ExternalWritable := 'False'} : Bool;
   // END_VAR
BEGIN
END_DATA_BLOCK

DATA_BLOCK "IEC_Timer_0_DB_134"   // DB208
{ S7_Optimized_Access := 'TRUE' }
// stored: InstanceOfName IEC_TIMER, OfSystemLibElement IEC_TIMER, OfSystemLibVersion 1.0
"IEC_TIMER"
   // VAR
   //    PT : Time;
   //    ET { ExternalWritable := 'False'} : Time;
   //    IN : Bool;
   //    Q { ExternalWritable := 'False'} : Bool;
   // END_VAR
BEGIN
END_DATA_BLOCK

DATA_BLOCK "IEC_Timer_0_DB_135"   // DB209
{ S7_Optimized_Access := 'TRUE' }
// stored: InstanceOfName IEC_TIMER, OfSystemLibElement IEC_TIMER, OfSystemLibVersion 1.0
"IEC_TIMER"
   // VAR
   //    PT : Time;
   //    ET { ExternalWritable := 'False'} : Time;
   //    IN : Bool;
   //    Q { ExternalWritable := 'False'} : Bool;
   // END_VAR
BEGIN
END_DATA_BLOCK

DATA_BLOCK "IEC_Timer_0_DB_136"   // DB210
{ S7_Optimized_Access := 'TRUE' }
// stored: InstanceOfName IEC_TIMER, OfSystemLibElement IEC_TIMER, OfSystemLibVersion 1.0
"IEC_TIMER"
   // VAR
   //    PT : Time;
   //    ET { ExternalWritable := 'False'} : Time;
   //    IN : Bool;
   //    Q { ExternalWritable := 'False'} : Bool;
   // END_VAR
BEGIN
END_DATA_BLOCK

DATA_BLOCK "IEC_Timer_0_DB_137"   // DB212
{ S7_Optimized_Access := 'TRUE' }
// stored: InstanceOfName IEC_TIMER, OfSystemLibElement IEC_TIMER, OfSystemLibVersion 1.0
"IEC_TIMER"
   // VAR
   //    PT : Time;
   //    ET { ExternalWritable := 'False'} : Time;
   //    IN : Bool;
   //    Q { ExternalWritable := 'False'} : Bool;
   // END_VAR
BEGIN
END_DATA_BLOCK

DATA_BLOCK "IEC_Timer_0_DB_14"   // DB36
{ S7_Optimized_Access := 'TRUE' }
// stored: InstanceOfName IEC_TIMER, OfSystemLibElement IEC_TIMER, OfSystemLibVersion 1.0
"IEC_TIMER"
   // VAR
   //    PT : Time;
   //    ET { ExternalWritable := 'False'} : Time;
   //    IN : Bool;
   //    Q { ExternalWritable := 'False'} : Bool;
   // END_VAR
BEGIN
END_DATA_BLOCK

DATA_BLOCK "IEC_Timer_0_DB_140"   // DB215
{ S7_Optimized_Access := 'TRUE' }
// stored: InstanceOfName IEC_TIMER, OfSystemLibElement IEC_TIMER, OfSystemLibVersion 1.0
"IEC_TIMER"
   // VAR
   //    PT : Time;
   //    ET { ExternalWritable := 'False'} : Time;
   //    IN : Bool;
   //    Q { ExternalWritable := 'False'} : Bool;
   // END_VAR
BEGIN
END_DATA_BLOCK

DATA_BLOCK "IEC_Timer_0_DB_141"   // DB216
{ S7_Optimized_Access := 'TRUE' }
// stored: InstanceOfName IEC_TIMER, OfSystemLibElement IEC_TIMER, OfSystemLibVersion 1.0
"IEC_TIMER"
   // VAR
   //    PT : Time;
   //    ET { ExternalWritable := 'False'} : Time;
   //    IN : Bool;
   //    Q { ExternalWritable := 'False'} : Bool;
   // END_VAR
BEGIN
END_DATA_BLOCK

DATA_BLOCK "IEC_Timer_0_DB_142"   // DB217
{ S7_Optimized_Access := 'TRUE' }
// stored: InstanceOfName IEC_TIMER, OfSystemLibElement IEC_TIMER, OfSystemLibVersion 1.0
"IEC_TIMER"
   // VAR
   //    PT : Time;
   //    ET { ExternalWritable := 'False'} : Time;
   //    IN : Bool;
   //    Q { ExternalWritable := 'False'} : Bool;
   // END_VAR
BEGIN
END_DATA_BLOCK

DATA_BLOCK "IEC_Timer_0_DB_143"   // DB218
{ S7_Optimized_Access := 'TRUE' }
// stored: InstanceOfName IEC_TIMER, OfSystemLibElement IEC_TIMER, OfSystemLibVersion 1.0
"IEC_TIMER"
   // VAR
   //    PT : Time;
   //    ET { ExternalWritable := 'False'} : Time;
   //    IN : Bool;
   //    Q { ExternalWritable := 'False'} : Bool;
   // END_VAR
BEGIN
END_DATA_BLOCK

DATA_BLOCK "IEC_Timer_0_DB_144"   // DB220
{ S7_Optimized_Access := 'TRUE' }
// stored: InstanceOfName IEC_TIMER, OfSystemLibElement IEC_TIMER, OfSystemLibVersion 1.0
"IEC_TIMER"
   // VAR
   //    PT : Time;
   //    ET { ExternalWritable := 'False'} : Time;
   //    IN : Bool;
   //    Q { ExternalWritable := 'False'} : Bool;
   // END_VAR
BEGIN
END_DATA_BLOCK

DATA_BLOCK "IEC_Timer_0_DB_145"   // DB221
{ S7_Optimized_Access := 'TRUE' }
// stored: InstanceOfName IEC_TIMER, OfSystemLibElement IEC_TIMER, OfSystemLibVersion 1.0
"IEC_TIMER"
   // VAR
   //    PT : Time;
   //    ET { ExternalWritable := 'False'} : Time;
   //    IN : Bool;
   //    Q { ExternalWritable := 'False'} : Bool;
   // END_VAR
BEGIN
END_DATA_BLOCK

DATA_BLOCK "IEC_Timer_0_DB_15"   // DB37
{ S7_Optimized_Access := 'TRUE' }
// stored: InstanceOfName IEC_TIMER, OfSystemLibElement IEC_TIMER, OfSystemLibVersion 1.0
"IEC_TIMER"
   // VAR
   //    PT : Time;
   //    ET { ExternalWritable := 'False'} : Time;
   //    IN : Bool;
   //    Q { ExternalWritable := 'False'} : Bool;
   // END_VAR
BEGIN
END_DATA_BLOCK

DATA_BLOCK "IEC_Timer_0_DB_16"   // DB39
{ S7_Optimized_Access := 'TRUE' }
// stored: InstanceOfName IEC_TIMER, OfSystemLibElement IEC_TIMER, OfSystemLibVersion 1.0
"IEC_TIMER"
   // VAR
   //    PT : Time;
   //    ET { ExternalWritable := 'False'} : Time;
   //    IN : Bool;
   //    Q { ExternalWritable := 'False'} : Bool;
   // END_VAR
BEGIN
END_DATA_BLOCK

DATA_BLOCK "IEC_Timer_0_DB_17"   // DB40
{ S7_Optimized_Access := 'TRUE' }
// stored: InstanceOfName IEC_TIMER, OfSystemLibElement IEC_TIMER, OfSystemLibVersion 1.0
"IEC_TIMER"
   // VAR
   //    PT : Time;
   //    ET { ExternalWritable := 'False'} : Time;
   //    IN : Bool;
   //    Q { ExternalWritable := 'False'} : Bool;
   // END_VAR
BEGIN
END_DATA_BLOCK

DATA_BLOCK "IEC_Timer_0_DB_18"   // DB59
{ S7_Optimized_Access := 'TRUE' }
// stored: InstanceOfName IEC_TIMER, OfSystemLibElement IEC_TIMER, OfSystemLibVersion 1.0
"IEC_TIMER"
   // VAR
   //    PT : Time;
   //    ET { ExternalWritable := 'False'} : Time;
   //    IN : Bool;
   //    Q { ExternalWritable := 'False'} : Bool;
   // END_VAR
BEGIN
END_DATA_BLOCK

DATA_BLOCK "IEC_Timer_0_DB_2"   // DB24
{ S7_Optimized_Access := 'TRUE' }
// stored: InstanceOfName IEC_TIMER, OfSystemLibElement IEC_TIMER, OfSystemLibVersion 1.0
"IEC_TIMER"
   // VAR
   //    PT : Time;
   //    ET { ExternalWritable := 'False'} : Time;
   //    IN : Bool;
   //    Q { ExternalWritable := 'False'} : Bool;
   // END_VAR
BEGIN
END_DATA_BLOCK

DATA_BLOCK "IEC_Timer_0_DB_20"   // DB61
{ S7_Optimized_Access := 'TRUE' }
// stored: InstanceOfName IEC_TIMER, OfSystemLibElement IEC_TIMER, OfSystemLibVersion 1.0
"IEC_TIMER"
   // VAR
   //    PT : Time;
   //    ET { ExternalWritable := 'False'} : Time;
   //    IN : Bool;
   //    Q { ExternalWritable := 'False'} : Bool;
   // END_VAR
BEGIN
END_DATA_BLOCK

DATA_BLOCK "IEC_Timer_0_DB_21"   // DB62
{ S7_Optimized_Access := 'TRUE' }
// stored: InstanceOfName IEC_TIMER, OfSystemLibElement IEC_TIMER, OfSystemLibVersion 1.0
"IEC_TIMER"
   // VAR
   //    PT : Time;
   //    ET { ExternalWritable := 'False'} : Time;
   //    IN : Bool;
   //    Q { ExternalWritable := 'False'} : Bool;
   // END_VAR
BEGIN
END_DATA_BLOCK

DATA_BLOCK "IEC_Timer_0_DB_22"   // DB63
{ S7_Optimized_Access := 'TRUE' }
// stored: InstanceOfName IEC_TIMER, OfSystemLibElement IEC_TIMER, OfSystemLibVersion 1.0
"IEC_TIMER"
   // VAR
   //    PT : Time;
   //    ET { ExternalWritable := 'False'} : Time;
   //    IN : Bool;
   //    Q { ExternalWritable := 'False'} : Bool;
   // END_VAR
BEGIN
END_DATA_BLOCK

DATA_BLOCK "IEC_Timer_0_DB_23"   // DB64
{ S7_Optimized_Access := 'TRUE' }
// stored: InstanceOfName IEC_TIMER, OfSystemLibElement IEC_TIMER, OfSystemLibVersion 1.0
"IEC_TIMER"
   // VAR
   //    PT : Time;
   //    ET { ExternalWritable := 'False'} : Time;
   //    IN : Bool;
   //    Q { ExternalWritable := 'False'} : Bool;
   // END_VAR
BEGIN
END_DATA_BLOCK

DATA_BLOCK "IEC_Timer_0_DB_24"   // DB65
{ S7_Optimized_Access := 'TRUE' }
// stored: InstanceOfName IEC_TIMER, OfSystemLibElement IEC_TIMER, OfSystemLibVersion 1.0
"IEC_TIMER"
   // VAR
   //    PT : Time;
   //    ET { ExternalWritable := 'False'} : Time;
   //    IN : Bool;
   //    Q { ExternalWritable := 'False'} : Bool;
   // END_VAR
BEGIN
END_DATA_BLOCK

DATA_BLOCK "IEC_Timer_0_DB_25"   // DB66
{ S7_Optimized_Access := 'TRUE' }
// stored: InstanceOfName IEC_TIMER, OfSystemLibElement IEC_TIMER, OfSystemLibVersion 1.0
"IEC_TIMER"
   // VAR
   //    PT : Time;
   //    ET { ExternalWritable := 'False'} : Time;
   //    IN : Bool;
   //    Q { ExternalWritable := 'False'} : Bool;
   // END_VAR
BEGIN
END_DATA_BLOCK

DATA_BLOCK "IEC_Timer_0_DB_26"   // DB67
{ S7_Optimized_Access := 'TRUE' }
// stored: InstanceOfName IEC_TIMER, OfSystemLibElement IEC_TIMER, OfSystemLibVersion 1.0
"IEC_TIMER"
   // VAR
   //    PT : Time;
   //    ET { ExternalWritable := 'False'} : Time;
   //    IN : Bool;
   //    Q { ExternalWritable := 'False'} : Bool;
   // END_VAR
BEGIN
END_DATA_BLOCK

DATA_BLOCK "IEC_Timer_0_DB_27"   // DB68
{ S7_Optimized_Access := 'TRUE' }
// stored: InstanceOfName IEC_TIMER, OfSystemLibElement IEC_TIMER, OfSystemLibVersion 1.0
"IEC_TIMER"
   // VAR
   //    PT : Time;
   //    ET { ExternalWritable := 'False'} : Time;
   //    IN : Bool;
   //    Q { ExternalWritable := 'False'} : Bool;
   // END_VAR
BEGIN
END_DATA_BLOCK

DATA_BLOCK "IEC_Timer_0_DB_28"   // DB69
{ S7_Optimized_Access := 'TRUE' }
// stored: InstanceOfName IEC_TIMER, OfSystemLibElement IEC_TIMER, OfSystemLibVersion 1.0
"IEC_TIMER"
   // VAR
   //    PT : Time;
   //    ET { ExternalWritable := 'False'} : Time;
   //    IN : Bool;
   //    Q { ExternalWritable := 'False'} : Bool;
   // END_VAR
BEGIN
END_DATA_BLOCK

DATA_BLOCK "IEC_Timer_0_DB_29"   // DB70
{ S7_Optimized_Access := 'TRUE' }
// stored: InstanceOfName IEC_TIMER, OfSystemLibElement IEC_TIMER, OfSystemLibVersion 1.0
"IEC_TIMER"
   // VAR
   //    PT : Time;
   //    ET { ExternalWritable := 'False'} : Time;
   //    IN : Bool;
   //    Q { ExternalWritable := 'False'} : Bool;
   // END_VAR
BEGIN
END_DATA_BLOCK

DATA_BLOCK "IEC_Timer_0_DB_3"   // DB25
{ S7_Optimized_Access := 'TRUE' }
// stored: InstanceOfName IEC_TIMER, OfSystemLibElement IEC_TIMER, OfSystemLibVersion 1.0
"IEC_TIMER"
   // VAR
   //    PT : Time;
   //    ET { ExternalWritable := 'False'} : Time;
   //    IN : Bool;
   //    Q { ExternalWritable := 'False'} : Bool;
   // END_VAR
BEGIN
END_DATA_BLOCK

DATA_BLOCK "IEC_Timer_0_DB_30"   // DB71
{ S7_Optimized_Access := 'TRUE' }
// stored: InstanceOfName IEC_TIMER, OfSystemLibElement IEC_TIMER, OfSystemLibVersion 1.0
"IEC_TIMER"
   // VAR
   //    PT : Time;
   //    ET { ExternalWritable := 'False'} : Time;
   //    IN : Bool;
   //    Q { ExternalWritable := 'False'} : Bool;
   // END_VAR
BEGIN
END_DATA_BLOCK

DATA_BLOCK "IEC_Timer_0_DB_31"   // DB72
{ S7_Optimized_Access := 'TRUE' }
// stored: InstanceOfName IEC_TIMER, OfSystemLibElement IEC_TIMER, OfSystemLibVersion 1.0
"IEC_TIMER"
   // VAR
   //    PT : Time;
   //    ET { ExternalWritable := 'False'} : Time;
   //    IN : Bool;
   //    Q { ExternalWritable := 'False'} : Bool;
   // END_VAR
BEGIN
END_DATA_BLOCK

DATA_BLOCK "IEC_Timer_0_DB_32"   // DB73
{ S7_Optimized_Access := 'TRUE' }
// stored: InstanceOfName IEC_TIMER, OfSystemLibElement IEC_TIMER, OfSystemLibVersion 1.0
"IEC_TIMER"
   // VAR
   //    PT : Time;
   //    ET { ExternalWritable := 'False'} : Time;
   //    IN : Bool;
   //    Q { ExternalWritable := 'False'} : Bool;
   // END_VAR
BEGIN
END_DATA_BLOCK

DATA_BLOCK "IEC_Timer_0_DB_33"   // DB74
{ S7_Optimized_Access := 'TRUE' }
// stored: InstanceOfName IEC_TIMER, OfSystemLibElement IEC_TIMER, OfSystemLibVersion 1.0
"IEC_TIMER"
   // VAR
   //    PT : Time;
   //    ET { ExternalWritable := 'False'} : Time;
   //    IN : Bool;
   //    Q { ExternalWritable := 'False'} : Bool;
   // END_VAR
BEGIN
END_DATA_BLOCK

DATA_BLOCK "IEC_Timer_0_DB_34"   // DB75
{ S7_Optimized_Access := 'TRUE' }
// stored: InstanceOfName IEC_TIMER, OfSystemLibElement IEC_TIMER, OfSystemLibVersion 1.0
"IEC_TIMER"
   // VAR
   //    PT : Time;
   //    ET { ExternalWritable := 'False'} : Time;
   //    IN : Bool;
   //    Q { ExternalWritable := 'False'} : Bool;
   // END_VAR
BEGIN
END_DATA_BLOCK

DATA_BLOCK "IEC_Timer_0_DB_35"   // DB79
{ S7_Optimized_Access := 'TRUE' }
// stored: InstanceOfName IEC_TIMER, OfSystemLibElement IEC_TIMER, OfSystemLibVersion 1.0
"IEC_TIMER"
   // VAR
   //    PT : Time;
   //    ET { ExternalWritable := 'False'} : Time;
   //    IN : Bool;
   //    Q { ExternalWritable := 'False'} : Bool;
   // END_VAR
BEGIN
END_DATA_BLOCK

DATA_BLOCK "IEC_Timer_0_DB_36"   // DB81
{ S7_Optimized_Access := 'TRUE' }
// stored: InstanceOfName IEC_TIMER, OfSystemLibElement IEC_TIMER, OfSystemLibVersion 1.0
"IEC_TIMER"
   // VAR
   //    PT : Time;
   //    ET { ExternalWritable := 'False'} : Time;
   //    IN : Bool;
   //    Q { ExternalWritable := 'False'} : Bool;
   // END_VAR
BEGIN
END_DATA_BLOCK

DATA_BLOCK "IEC_Timer_0_DB_37"   // DB104
{ S7_Optimized_Access := 'TRUE' }
// stored: InstanceOfName IEC_TIMER, OfSystemLibElement IEC_TIMER, OfSystemLibVersion 1.0
"IEC_TIMER"
   // VAR
   //    PT : Time;
   //    ET { ExternalWritable := 'False'} : Time;
   //    IN : Bool;
   //    Q { ExternalWritable := 'False'} : Bool;
   // END_VAR
BEGIN
END_DATA_BLOCK

DATA_BLOCK "IEC_Timer_0_DB_38"   // DB111
{ S7_Optimized_Access := 'TRUE' }
// stored: InstanceOfName IEC_TIMER, OfSystemLibElement IEC_TIMER, OfSystemLibVersion 1.0
"IEC_TIMER"
   // VAR
   //    PT : Time;
   //    ET { ExternalWritable := 'False'} : Time;
   //    IN : Bool;
   //    Q { ExternalWritable := 'False'} : Bool;
   // END_VAR
BEGIN
END_DATA_BLOCK

DATA_BLOCK "IEC_Timer_0_DB_39"   // DB84
{ S7_Optimized_Access := 'TRUE' }
// stored: InstanceOfName IEC_TIMER, OfSystemLibElement IEC_TIMER, OfSystemLibVersion 1.0
"IEC_TIMER"
   // VAR
   //    PT : Time;
   //    ET { ExternalWritable := 'False'} : Time;
   //    IN : Bool;
   //    Q { ExternalWritable := 'False'} : Bool;
   // END_VAR
BEGIN
END_DATA_BLOCK

DATA_BLOCK "IEC_Timer_0_DB_4"   // DB26
{ S7_Optimized_Access := 'TRUE' }
// stored: InstanceOfName IEC_TIMER, OfSystemLibElement IEC_TIMER, OfSystemLibVersion 1.0
"IEC_TIMER"
   // VAR
   //    PT : Time;
   //    ET { ExternalWritable := 'False'} : Time;
   //    IN : Bool;
   //    Q { ExternalWritable := 'False'} : Bool;
   // END_VAR
BEGIN
END_DATA_BLOCK

DATA_BLOCK "IEC_Timer_0_DB_40"   // DB85
{ S7_Optimized_Access := 'TRUE' }
// stored: InstanceOfName IEC_TIMER, OfSystemLibElement IEC_TIMER, OfSystemLibVersion 1.0
"IEC_TIMER"
   // VAR
   //    PT : Time;
   //    ET { ExternalWritable := 'False'} : Time;
   //    IN : Bool;
   //    Q { ExternalWritable := 'False'} : Bool;
   // END_VAR
BEGIN
END_DATA_BLOCK

DATA_BLOCK "IEC_Timer_0_DB_41"   // DB86
{ S7_Optimized_Access := 'TRUE' }
// stored: InstanceOfName IEC_TIMER, OfSystemLibElement IEC_TIMER, OfSystemLibVersion 1.0
"IEC_TIMER"
   // VAR
   //    PT : Time;
   //    ET { ExternalWritable := 'False'} : Time;
   //    IN : Bool;
   //    Q { ExternalWritable := 'False'} : Bool;
   // END_VAR
BEGIN
END_DATA_BLOCK

DATA_BLOCK "IEC_Timer_0_DB_42"   // DB87
{ S7_Optimized_Access := 'TRUE' }
// stored: InstanceOfName IEC_TIMER, OfSystemLibElement IEC_TIMER, OfSystemLibVersion 1.0
"IEC_TIMER"
   // VAR
   //    PT : Time;
   //    ET { ExternalWritable := 'False'} : Time;
   //    IN : Bool;
   //    Q { ExternalWritable := 'False'} : Bool;
   // END_VAR
BEGIN
END_DATA_BLOCK

DATA_BLOCK "IEC_Timer_0_DB_43"   // DB88
{ S7_Optimized_Access := 'TRUE' }
// stored: InstanceOfName IEC_TIMER, OfSystemLibElement IEC_TIMER, OfSystemLibVersion 1.0
"IEC_TIMER"
   // VAR
   //    PT : Time;
   //    ET { ExternalWritable := 'False'} : Time;
   //    IN : Bool;
   //    Q { ExternalWritable := 'False'} : Bool;
   // END_VAR
BEGIN
END_DATA_BLOCK

DATA_BLOCK "IEC_Timer_0_DB_44"   // DB89
{ S7_Optimized_Access := 'TRUE' }
// stored: InstanceOfName IEC_TIMER, OfSystemLibElement IEC_TIMER, OfSystemLibVersion 1.0
"IEC_TIMER"
   // VAR
   //    PT : Time;
   //    ET { ExternalWritable := 'False'} : Time;
   //    IN : Bool;
   //    Q { ExternalWritable := 'False'} : Bool;
   // END_VAR
BEGIN
END_DATA_BLOCK

DATA_BLOCK "IEC_Timer_0_DB_45"   // DB113
{ S7_Optimized_Access := 'TRUE' }
// stored: InstanceOfName IEC_TIMER, OfSystemLibElement IEC_TIMER, OfSystemLibVersion 1.0
"IEC_TIMER"
   // VAR
   //    PT : Time;
   //    ET { ExternalWritable := 'False'} : Time;
   //    IN : Bool;
   //    Q { ExternalWritable := 'False'} : Bool;
   // END_VAR
BEGIN
END_DATA_BLOCK

DATA_BLOCK "IEC_Timer_0_DB_46"   // DB91
{ S7_Optimized_Access := 'TRUE' }
// stored: InstanceOfName IEC_TIMER, OfSystemLibElement IEC_TIMER, OfSystemLibVersion 1.0
"IEC_TIMER"
   // VAR
   //    PT : Time;
   //    ET { ExternalWritable := 'False'} : Time;
   //    IN : Bool;
   //    Q { ExternalWritable := 'False'} : Bool;
   // END_VAR
BEGIN
END_DATA_BLOCK

DATA_BLOCK "IEC_Timer_0_DB_47"   // DB92
{ S7_Optimized_Access := 'TRUE' }
// stored: InstanceOfName IEC_TIMER, OfSystemLibElement IEC_TIMER, OfSystemLibVersion 1.0
"IEC_TIMER"
   // VAR
   //    PT : Time;
   //    ET { ExternalWritable := 'False'} : Time;
   //    IN : Bool;
   //    Q { ExternalWritable := 'False'} : Bool;
   // END_VAR
BEGIN
END_DATA_BLOCK

DATA_BLOCK "IEC_Timer_0_DB_48"   // DB93
{ S7_Optimized_Access := 'TRUE' }
// stored: InstanceOfName IEC_TIMER, OfSystemLibElement IEC_TIMER, OfSystemLibVersion 1.0
"IEC_TIMER"
   // VAR
   //    PT : Time;
   //    ET { ExternalWritable := 'False'} : Time;
   //    IN : Bool;
   //    Q { ExternalWritable := 'False'} : Bool;
   // END_VAR
BEGIN
END_DATA_BLOCK

DATA_BLOCK "IEC_Timer_0_DB_49"   // DB94
{ S7_Optimized_Access := 'TRUE' }
// stored: InstanceOfName IEC_TIMER, OfSystemLibElement IEC_TIMER, OfSystemLibVersion 1.0
"IEC_TIMER"
   // VAR
   //    PT : Time;
   //    ET { ExternalWritable := 'False'} : Time;
   //    IN : Bool;
   //    Q { ExternalWritable := 'False'} : Bool;
   // END_VAR
BEGIN
END_DATA_BLOCK

DATA_BLOCK "IEC_Timer_0_DB_5"   // DB27
{ S7_Optimized_Access := 'TRUE' }
// stored: InstanceOfName IEC_TIMER, OfSystemLibElement IEC_TIMER, OfSystemLibVersion 1.0
"IEC_TIMER"
   // VAR
   //    PT : Time;
   //    ET { ExternalWritable := 'False'} : Time;
   //    IN : Bool;
   //    Q { ExternalWritable := 'False'} : Bool;
   // END_VAR
BEGIN
END_DATA_BLOCK

DATA_BLOCK "IEC_Timer_0_DB_50"   // DB95
{ S7_Optimized_Access := 'TRUE' }
// stored: InstanceOfName IEC_TIMER, OfSystemLibElement IEC_TIMER, OfSystemLibVersion 1.0
"IEC_TIMER"
   // VAR
   //    PT : Time;
   //    ET { ExternalWritable := 'False'} : Time;
   //    IN : Bool;
   //    Q { ExternalWritable := 'False'} : Bool;
   // END_VAR
BEGIN
END_DATA_BLOCK

DATA_BLOCK "IEC_Timer_0_DB_51"   // DB96
{ S7_Optimized_Access := 'TRUE' }
// stored: InstanceOfName IEC_TIMER, OfSystemLibElement IEC_TIMER, OfSystemLibVersion 1.0
"IEC_TIMER"
   // VAR
   //    PT : Time;
   //    ET { ExternalWritable := 'False'} : Time;
   //    IN : Bool;
   //    Q { ExternalWritable := 'False'} : Bool;
   // END_VAR
BEGIN
END_DATA_BLOCK

DATA_BLOCK "IEC_Timer_0_DB_52"   // DB97
{ S7_Optimized_Access := 'TRUE' }
// stored: InstanceOfName IEC_TIMER, OfSystemLibElement IEC_TIMER, OfSystemLibVersion 1.0
"IEC_TIMER"
   // VAR
   //    PT : Time;
   //    ET { ExternalWritable := 'False'} : Time;
   //    IN : Bool;
   //    Q { ExternalWritable := 'False'} : Bool;
   // END_VAR
BEGIN
END_DATA_BLOCK

DATA_BLOCK "IEC_Timer_0_DB_53"   // DB98
{ S7_Optimized_Access := 'TRUE' }
// stored: InstanceOfName IEC_TIMER, OfSystemLibElement IEC_TIMER, OfSystemLibVersion 1.0
"IEC_TIMER"
   // VAR
   //    PT : Time;
   //    ET { ExternalWritable := 'False'} : Time;
   //    IN : Bool;
   //    Q { ExternalWritable := 'False'} : Bool;
   // END_VAR
BEGIN
END_DATA_BLOCK

DATA_BLOCK "IEC_Timer_0_DB_54"   // DB99
{ S7_Optimized_Access := 'TRUE' }
// stored: InstanceOfName IEC_TIMER, OfSystemLibElement IEC_TIMER, OfSystemLibVersion 1.0
"IEC_TIMER"
   // VAR
   //    PT : Time;
   //    ET { ExternalWritable := 'False'} : Time;
   //    IN : Bool;
   //    Q { ExternalWritable := 'False'} : Bool;
   // END_VAR
BEGIN
END_DATA_BLOCK

DATA_BLOCK "IEC_Timer_0_DB_55"   // DB100
{ S7_Optimized_Access := 'TRUE' }
// stored: InstanceOfName IEC_TIMER, OfSystemLibElement IEC_TIMER, OfSystemLibVersion 1.0
"IEC_TIMER"
   // VAR
   //    PT : Time;
   //    ET { ExternalWritable := 'False'} : Time;
   //    IN : Bool;
   //    Q { ExternalWritable := 'False'} : Bool;
   // END_VAR
BEGIN
END_DATA_BLOCK

DATA_BLOCK "IEC_Timer_0_DB_56"   // DB101
{ S7_Optimized_Access := 'TRUE' }
// stored: InstanceOfName IEC_TIMER, OfSystemLibElement IEC_TIMER, OfSystemLibVersion 1.0
"IEC_TIMER"
   // VAR
   //    PT : Time;
   //    ET { ExternalWritable := 'False'} : Time;
   //    IN : Bool;
   //    Q { ExternalWritable := 'False'} : Bool;
   // END_VAR
BEGIN
END_DATA_BLOCK

DATA_BLOCK "IEC_Timer_0_DB_57"   // DB102
{ S7_Optimized_Access := 'TRUE' }
// stored: InstanceOfName IEC_TIMER, OfSystemLibElement IEC_TIMER, OfSystemLibVersion 1.0
"IEC_TIMER"
   // VAR
   //    PT : Time;
   //    ET { ExternalWritable := 'False'} : Time;
   //    IN : Bool;
   //    Q { ExternalWritable := 'False'} : Bool;
   // END_VAR
BEGIN
END_DATA_BLOCK

DATA_BLOCK "IEC_Timer_0_DB_58"   // DB103
{ S7_Optimized_Access := 'TRUE' }
// stored: InstanceOfName IEC_TIMER, OfSystemLibElement IEC_TIMER, OfSystemLibVersion 1.0
"IEC_TIMER"
   // VAR
   //    PT : Time;
   //    ET { ExternalWritable := 'False'} : Time;
   //    IN : Bool;
   //    Q { ExternalWritable := 'False'} : Bool;
   // END_VAR
BEGIN
END_DATA_BLOCK

DATA_BLOCK "IEC_Timer_0_DB_59"   // DB110
{ S7_Optimized_Access := 'TRUE' }
// stored: InstanceOfName IEC_TIMER, OfSystemLibElement IEC_TIMER, OfSystemLibVersion 1.0
"IEC_TIMER"
   // VAR
   //    PT : Time;
   //    ET { ExternalWritable := 'False'} : Time;
   //    IN : Bool;
   //    Q { ExternalWritable := 'False'} : Bool;
   // END_VAR
BEGIN
END_DATA_BLOCK

DATA_BLOCK "IEC_Timer_0_DB_6"   // DB28
{ S7_Optimized_Access := 'TRUE' }
// stored: InstanceOfName IEC_TIMER, OfSystemLibElement IEC_TIMER, OfSystemLibVersion 1.0
"IEC_TIMER"
   // VAR
   //    PT : Time;
   //    ET { ExternalWritable := 'False'} : Time;
   //    IN : Bool;
   //    Q { ExternalWritable := 'False'} : Bool;
   // END_VAR
BEGIN
END_DATA_BLOCK

DATA_BLOCK "IEC_Timer_0_DB_60"   // DB114
{ S7_Optimized_Access := 'TRUE' }
// stored: InstanceOfName IEC_TIMER, OfSystemLibElement IEC_TIMER, OfSystemLibVersion 1.0
"IEC_TIMER"
   // VAR
   //    PT : Time;
   //    ET { ExternalWritable := 'False'} : Time;
   //    IN : Bool;
   //    Q { ExternalWritable := 'False'} : Bool;
   // END_VAR
BEGIN
END_DATA_BLOCK

DATA_BLOCK "IEC_Timer_0_DB_61"   // DB115
{ S7_Optimized_Access := 'TRUE' }
// stored: InstanceOfName IEC_TIMER, OfSystemLibElement IEC_TIMER, OfSystemLibVersion 1.0
"IEC_TIMER"
   // VAR
   //    PT : Time;
   //    ET { ExternalWritable := 'False'} : Time;
   //    IN : Bool;
   //    Q { ExternalWritable := 'False'} : Bool;
   // END_VAR
BEGIN
END_DATA_BLOCK

DATA_BLOCK "IEC_Timer_0_DB_62"   // DB117
{ S7_Optimized_Access := 'TRUE' }
// stored: InstanceOfName IEC_TIMER, OfSystemLibElement IEC_TIMER, OfSystemLibVersion 1.0
"IEC_TIMER"
   // VAR
   //    PT : Time;
   //    ET { ExternalWritable := 'False'} : Time;
   //    IN : Bool;
   //    Q { ExternalWritable := 'False'} : Bool;
   // END_VAR
BEGIN
END_DATA_BLOCK

DATA_BLOCK "IEC_Timer_0_DB_63"   // DB118
{ S7_Optimized_Access := 'TRUE' }
// stored: InstanceOfName IEC_TIMER, OfSystemLibElement IEC_TIMER, OfSystemLibVersion 1.0
"IEC_TIMER"
   // VAR
   //    PT : Time;
   //    ET { ExternalWritable := 'False'} : Time;
   //    IN : Bool;
   //    Q { ExternalWritable := 'False'} : Bool;
   // END_VAR
BEGIN
END_DATA_BLOCK

DATA_BLOCK "IEC_Timer_0_DB_64"   // DB120
{ S7_Optimized_Access := 'TRUE' }
// stored: InstanceOfName IEC_TIMER, OfSystemLibElement IEC_TIMER, OfSystemLibVersion 1.0
"IEC_TIMER"
   // VAR
   //    PT : Time;
   //    ET { ExternalWritable := 'False'} : Time;
   //    IN : Bool;
   //    Q { ExternalWritable := 'False'} : Bool;
   // END_VAR
BEGIN
END_DATA_BLOCK

DATA_BLOCK "IEC_Timer_0_DB_65"   // DB121
{ S7_Optimized_Access := 'TRUE' }
// stored: InstanceOfName IEC_TIMER, OfSystemLibElement IEC_TIMER, OfSystemLibVersion 1.0
"IEC_TIMER"
   // VAR
   //    PT : Time;
   //    ET { ExternalWritable := 'False'} : Time;
   //    IN : Bool;
   //    Q { ExternalWritable := 'False'} : Bool;
   // END_VAR
BEGIN
END_DATA_BLOCK

DATA_BLOCK "IEC_Timer_0_DB_66"   // DB123
{ S7_Optimized_Access := 'TRUE' }
// stored: InstanceOfName IEC_TIMER, OfSystemLibElement IEC_TIMER, OfSystemLibVersion 1.0
"IEC_TIMER"
   // VAR
   //    PT : Time;
   //    ET { ExternalWritable := 'False'} : Time;
   //    IN : Bool;
   //    Q { ExternalWritable := 'False'} : Bool;
   // END_VAR
BEGIN
END_DATA_BLOCK

DATA_BLOCK "IEC_Timer_0_DB_67"   // DB125
{ S7_Optimized_Access := 'TRUE' }
// stored: InstanceOfName IEC_TIMER, OfSystemLibElement IEC_TIMER, OfSystemLibVersion 1.0
"IEC_TIMER"
   // VAR
   //    PT : Time;
   //    ET { ExternalWritable := 'False'} : Time;
   //    IN : Bool;
   //    Q { ExternalWritable := 'False'} : Bool;
   // END_VAR
BEGIN
END_DATA_BLOCK

DATA_BLOCK "IEC_Timer_0_DB_68"   // DB223
{ S7_Optimized_Access := 'TRUE' }
// stored: InstanceOfName IEC_TIMER, OfSystemLibElement IEC_TIMER, OfSystemLibVersion 1.0
"IEC_TIMER"
   // VAR
   //    PT : Time;
   //    ET { ExternalWritable := 'False'} : Time;
   //    IN : Bool;
   //    Q { ExternalWritable := 'False'} : Bool;
   // END_VAR
BEGIN
END_DATA_BLOCK

DATA_BLOCK "IEC_Timer_0_DB_69"   // DB127
{ S7_Optimized_Access := 'TRUE' }
// stored: InstanceOfName IEC_TIMER, OfSystemLibElement IEC_TIMER, OfSystemLibVersion 1.0
"IEC_TIMER"
   // VAR
   //    PT : Time;
   //    ET { ExternalWritable := 'False'} : Time;
   //    IN : Bool;
   //    Q { ExternalWritable := 'False'} : Bool;
   // END_VAR
BEGIN
END_DATA_BLOCK

DATA_BLOCK "IEC_Timer_0_DB_7"   // DB29
{ S7_Optimized_Access := 'TRUE' }
// stored: InstanceOfName IEC_TIMER, OfSystemLibElement IEC_TIMER, OfSystemLibVersion 1.0
"IEC_TIMER"
   // VAR
   //    PT : Time;
   //    ET { ExternalWritable := 'False'} : Time;
   //    IN : Bool;
   //    Q { ExternalWritable := 'False'} : Bool;
   // END_VAR
BEGIN
END_DATA_BLOCK

DATA_BLOCK "IEC_Timer_0_DB_70"   // DB129
{ S7_Optimized_Access := 'TRUE' }
// stored: InstanceOfName IEC_TIMER, OfSystemLibElement IEC_TIMER, OfSystemLibVersion 1.0
"IEC_TIMER"
   // VAR
   //    PT : Time;
   //    ET { ExternalWritable := 'False'} : Time;
   //    IN : Bool;
   //    Q { ExternalWritable := 'False'} : Bool;
   // END_VAR
BEGIN
END_DATA_BLOCK

DATA_BLOCK "IEC_Timer_0_DB_71"   // DB130
{ S7_Optimized_Access := 'TRUE' }
// stored: InstanceOfName IEC_TIMER, OfSystemLibElement IEC_TIMER, OfSystemLibVersion 1.0
"IEC_TIMER"
   // VAR
   //    PT : Time;
   //    ET { ExternalWritable := 'False'} : Time;
   //    IN : Bool;
   //    Q { ExternalWritable := 'False'} : Bool;
   // END_VAR
BEGIN
END_DATA_BLOCK

DATA_BLOCK "IEC_Timer_0_DB_72"   // DB132
{ S7_Optimized_Access := 'TRUE' }
// stored: InstanceOfName IEC_TIMER, OfSystemLibElement IEC_TIMER, OfSystemLibVersion 1.0
"IEC_TIMER"
   // VAR
   //    PT : Time;
   //    ET { ExternalWritable := 'False'} : Time;
   //    IN : Bool;
   //    Q { ExternalWritable := 'False'} : Bool;
   // END_VAR
BEGIN
END_DATA_BLOCK

DATA_BLOCK "IEC_Timer_0_DB_73"   // DB133
{ S7_Optimized_Access := 'TRUE' }
// stored: InstanceOfName IEC_TIMER, OfSystemLibElement IEC_TIMER, OfSystemLibVersion 1.0
"IEC_TIMER"
   // VAR
   //    PT : Time;
   //    ET { ExternalWritable := 'False'} : Time;
   //    IN : Bool;
   //    Q { ExternalWritable := 'False'} : Bool;
   // END_VAR
BEGIN
END_DATA_BLOCK

DATA_BLOCK "IEC_Timer_0_DB_74"   // DB228
{ S7_Optimized_Access := 'TRUE' }
// stored: InstanceOfName IEC_TIMER, OfSystemLibElement IEC_TIMER, OfSystemLibVersion 1.0
"IEC_TIMER"
   // VAR
   //    PT : Time;
   //    ET { ExternalWritable := 'False'} : Time;
   //    IN : Bool;
   //    Q { ExternalWritable := 'False'} : Bool;
   // END_VAR
BEGIN
END_DATA_BLOCK

DATA_BLOCK "IEC_Timer_0_DB_75"   // DB230
{ S7_Optimized_Access := 'TRUE' }
// stored: InstanceOfName IEC_TIMER, OfSystemLibElement IEC_TIMER, OfSystemLibVersion 1.0
"IEC_TIMER"
   // VAR
   //    PT : Time;
   //    ET { ExternalWritable := 'False'} : Time;
   //    IN : Bool;
   //    Q { ExternalWritable := 'False'} : Bool;
   // END_VAR
BEGIN
END_DATA_BLOCK

DATA_BLOCK "IEC_Timer_0_DB_76"   // DB137
{ S7_Optimized_Access := 'TRUE' }
// stored: InstanceOfName IEC_TIMER, OfSystemLibElement IEC_TIMER, OfSystemLibVersion 1.0
"IEC_TIMER"
   // VAR
   //    PT : Time;
   //    ET { ExternalWritable := 'False'} : Time;
   //    IN : Bool;
   //    Q { ExternalWritable := 'False'} : Bool;
   // END_VAR
BEGIN
END_DATA_BLOCK

DATA_BLOCK "IEC_Timer_0_DB_77"   // DB138
{ S7_Optimized_Access := 'TRUE' }
// stored: InstanceOfName IEC_TIMER, OfSystemLibElement IEC_TIMER, OfSystemLibVersion 1.0
"IEC_TIMER"
   // VAR
   //    PT : Time;
   //    ET { ExternalWritable := 'False'} : Time;
   //    IN : Bool;
   //    Q { ExternalWritable := 'False'} : Bool;
   // END_VAR
BEGIN
END_DATA_BLOCK

DATA_BLOCK "IEC_Timer_0_DB_78"   // DB139
{ S7_Optimized_Access := 'TRUE' }
// stored: InstanceOfName IEC_TIMER, OfSystemLibElement IEC_TIMER, OfSystemLibVersion 1.0
"IEC_TIMER"
   // VAR
   //    PT : Time;
   //    ET { ExternalWritable := 'False'} : Time;
   //    IN : Bool;
   //    Q { ExternalWritable := 'False'} : Bool;
   // END_VAR
BEGIN
END_DATA_BLOCK

DATA_BLOCK "IEC_Timer_0_DB_79"   // DB140
{ S7_Optimized_Access := 'TRUE' }
// stored: InstanceOfName IEC_TIMER, OfSystemLibElement IEC_TIMER, OfSystemLibVersion 1.0
"IEC_TIMER"
   // VAR
   //    PT : Time;
   //    ET { ExternalWritable := 'False'} : Time;
   //    IN : Bool;
   //    Q { ExternalWritable := 'False'} : Bool;
   // END_VAR
BEGIN
END_DATA_BLOCK

DATA_BLOCK "IEC_Timer_0_DB_8"   // DB30
{ S7_Optimized_Access := 'TRUE' }
// stored: InstanceOfName IEC_TIMER, OfSystemLibElement IEC_TIMER, OfSystemLibVersion 1.0
"IEC_TIMER"
   // VAR
   //    PT : Time;
   //    ET { ExternalWritable := 'False'} : Time;
   //    IN : Bool;
   //    Q { ExternalWritable := 'False'} : Bool;
   // END_VAR
BEGIN
END_DATA_BLOCK

DATA_BLOCK "IEC_Timer_0_DB_80"   // DB141
{ S7_Optimized_Access := 'TRUE' }
// stored: InstanceOfName IEC_TIMER, OfSystemLibElement IEC_TIMER, OfSystemLibVersion 1.0
"IEC_TIMER"
   // VAR
   //    PT : Time;
   //    ET { ExternalWritable := 'False'} : Time;
   //    IN : Bool;
   //    Q { ExternalWritable := 'False'} : Bool;
   // END_VAR
BEGIN
END_DATA_BLOCK

DATA_BLOCK "IEC_Timer_0_DB_81"   // DB142
{ S7_Optimized_Access := 'TRUE' }
// stored: InstanceOfName IEC_TIMER, OfSystemLibElement IEC_TIMER, OfSystemLibVersion 1.0
"IEC_TIMER"
   // VAR
   //    PT : Time;
   //    ET { ExternalWritable := 'False'} : Time;
   //    IN : Bool;
   //    Q { ExternalWritable := 'False'} : Bool;
   // END_VAR
BEGIN
END_DATA_BLOCK

